KUKA KRL program: EPS_2_25694_BP03_A_20251120043254.src

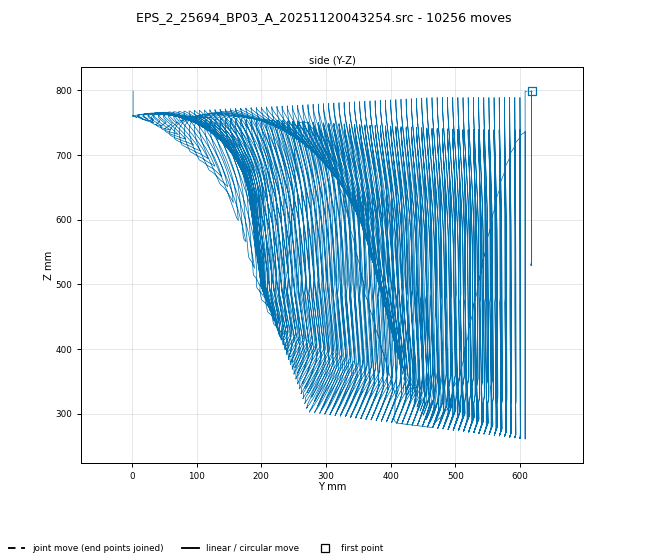
[picture p0: tool path of EPS_2_25694_BP03_A_20251120043254.src, 10256 of 10258 moves have a stored position in this frame; points joined in program order, loops and branches not executed]
&ACCESS RVP
&REL 4
&COMMENT QRS 19112012
&PARAM EDITMASK = *
DEF PART()
EXT BAS (BAS_COMMAND :IN,REAL :IN )
INT I
BAS (#INITMOV,0 )

;KUKA QRS Post kuka4.cps  Date:22-06-2017 !

File_ID=2919

QRS_PRE_INIT()

;Init var - Until changes are made in qrs_pre_init
Outlet_Square_prg=0
Inlet_1_Square_prg=0
Inlet_2_Square_prg=0
Inlet_3_Square_prg=0
Inlet_4_Square_prg=0
Inlet_5_Square_prg=0

Outlet_1={X 0.000, Y 466.000, Z 560.500, B 0.000, E1 0.000 }
Inlet_1={X 0.000, Y 466.000, Z 548.500, B 0.000, E1 90.000 }
Inlet_2={X 0.000, Y 519.840, Z 613.500, B 0.000, E1 205.000 }
Outlet_1_type=457
Inlet_1_type=381
Inlet_2_type=251
;QRS#1=Sidecore dimensions
;QRS#2=450-18" Concrete
;QRS#3=375-15" Concrete
;QRS#4=250-10" PVC SDR 35
;QRS#5=
;QRS#6=
;QRS#7=
;QRS#8=
;QRS#9=28A PSX-2
;QRS#10=24L PSX-2
;QRS#11=14M PSX
;QRS#12=
;QRS#13=
;QRS#14=
;QRS#15=
;QRS#16=1220x127x1143 3,75'
;QRS#17=EPS Height
;QRS#18=789
;QRS#19=*
;QRS#20= UPDATED VERSION 22-06-2017
;QRS#21=*
Outlet_Square=0250
Inlet_1_Square=0150
Inlet_2_Square=0100
Inlet_3_Square=0
Inlet_4_Square=0
Inlet_5_Square=0
Mill_Square=1
Outlet_Square_Prg=274
Inlet_1_Square_prg=261
Inlet_2_Square_prg=205

QRS_INIT()

$ADVANCE=5

; T1
PTP {E1 170.917,E2 170.917}
PTP {X 0,Y 617.926,A -85,B 0,C 180,E1 170.917,E2 170.917,E3 0,E4 0,E5 0,E6 0}
QRS_SPEED_INIT()
LIN {X 0,Y 617.926,Z 799,A -85,B 0,C 180,E1 170.917,E2 170.917,E3 0,E4 0,E5 0,E6 0} C_VEL
LIN {X 0,Y 617.926,Z 732.08,A -85,B 0,C 180,E1 170.917,E2 170.917} C_VEL
LIN {X 0,Y 617.926,Z 723.896,A -85,B 0,C 180,E1 170.917,E2 170.917} C_VEL
LIN {X 0,Y 617.92,Z 722.066,A -85,B 0,C 180,E1 171.177,E2 171.177} C_VEL
LIN {X 0,Y 617.969,Z 725.43,A -85,B 0,C 180,E1 171.885,E2 171.885} C_VEL
LIN {X 0,Y 617.858,Z 729.365,A -85,B 0,C 180,E1 172.817,E2 172.817} C_VEL
LIN {X 0,Y 617.844,Z 732.739,A -85,B 0,C 180,E1 173.747,E2 173.747} C_VEL
LIN {X 0,Y 617.965,Z 735.568,A -85,B 0,C 180,E1 174.678,E2 174.678} C_VEL
LIN {X 0,Y 617.921,Z 737.95,A -85,B 0,C 180,E1 175.605,E2 175.605} C_VEL
LIN {X 0,Y 617.836,Z 739.867,A -85,B 0,C 180,E1 176.531,E2 176.531} C_VEL
LIN {X 0,Y 617.889,Z 741.283,A -85,B 0,C 180,E1 177.457,E2 177.457} C_VEL
LIN {X 0,Y 617.913,Z 742.583,A -85,B 0,C 180,E1 178.844,E2 178.844} C_VEL
LIN {X 0,Y 617.836,Z 742.919,A -85,B 0,C 180,E1 179.769,E2 179.769} C_VEL
LIN {X 0,Y 617.896,Z 742.773,A -85,B 0,C 180,E1 180.693,E2 180.693} C_VEL
LIN {X 0,Y 617.953,Z 742.507,A -85,B 0,C 180,E1 181.155,E2 181.155} C_VEL
LIN {X 0,Y 617.906,Z 741.719,A -85,B 0,C 180,E1 182.08,E2 182.08} C_VEL
LIN {X 0,Y 617.845,Z 741.189,A -85,B 0,C 180,E1 182.543,E2 182.543} C_VEL
LIN {X 0,Y 617.837,Z 739.718,A -85,B 0,C 180,E1 183.469,E2 183.469} C_VEL
LIN {X 0,Y 617.952,Z 737.748,A -85,B 0,C 180,E1 184.395,E2 184.395} C_VEL
LIN {X 0,Y 617.906,Z 735.343,A -85,B 0,C 180,E1 185.323,E2 185.323} C_VEL
LIN {X 0,Y 617.823,Z 732.457,A -85,B 0,C 180,E1 186.253,E2 186.253} C_VEL
LIN {X 0,Y 617.893,Z 729.022,A -85,B 0,C 180,E1 187.183,E2 187.183} C_VEL
LIN {X 0,Y 617.971,Z 725.042,A -85,B 0,C 180,E1 188.115,E2 188.115} C_VEL
LIN {X 0,Y 617.879,Z 720.318,A -85,B 0,C 180,E1 189.086,E2 189.086} C_VEL
LIN {X 0,Y 617.904,Z 714.839,A -85,B 0,C 180,E1 190.065,E2 190.065} C_VEL
LIN {X 0,Y 617.99,Z 710.607,A -85,B 0,C 180,E1 190.75,E2 190.75} C_VEL
LIN {X 0,Y 617.939,Z 704.579,A -85,B 0,C 180,E1 191.634,E2 191.634} C_VEL
LIN {X 0,Y 617.924,Z 699.032,A -85,B 0,C 180,E1 192.373,E2 192.373} C_VEL
LIN {X 0,Y 617.977,Z 692.923,A -85,B 0,C 180,E1 193.112,E2 193.112} C_VEL
LIN {X 0,Y 617.99,Z 686.213,A -85,B 0,C 180,E1 193.854,E2 193.854} C_VEL
LIN {X 0,Y 617.953,Z 678.824,A -85,B 0,C 180,E1 194.6,E2 194.6} C_VEL
LIN {X 0,Y 617.973,Z 671.228,A -85,B 0,C 180,E1 195.296,E2 195.296} C_VEL
LIN {X 0,Y 617.987,Z 664.189,A -85,B 0,C 180,E1 195.886,E2 195.886} C_VEL
LIN {X 0,Y 617.986,Z 657.726,A -85,B 0,C 180,E1 196.388,E2 196.388} C_VEL
LIN {X 0,Y 617.976,Z 650.68,A -85,B 0,C 180,E1 196.894,E2 196.894} C_VEL
LIN {X 0,Y 617.993,Z 642.968,A -85,B 0,C 180,E1 197.402,E2 197.402} C_VEL
LIN {X 0,Y 617.989,Z 634.017,A -85,B 0,C 180,E1 197.935,E2 197.935} C_VEL
LIN {X 0,Y 618.005,Z 624.088,A -85,B 0,C 180,E1 198.462,E2 198.462} C_VEL
LIN {X 0,Y 617.991,Z 616.381,A -85,B 0,C 180,E1 198.833,E2 198.833} C_VEL
LIN {X 0,Y 617.89,Z 606.2,A -85,B 0,C 180,E1 199.269,E2 199.269} C_VEL
LIN {X 0,Y 617.965,Z 596.887,A -85,B 0,C 180,E1 199.613,E2 199.613} C_VEL
LIN {X 0,Y 617.956,Z 586.341,A -85,B 0,C 180,E1 199.95,E2 199.95} C_VEL
LIN {X 0,Y 617.862,Z 577.249,A -85,B 0,C 180,E1 200.201,E2 200.201} C_VEL
LIN {X 0,Y 617.986,Z 567.625,A -85,B 0,C 180,E1 200.414,E2 200.414} C_VEL
LIN {X 0,Y 618.002,Z 557.725,A -85,B 0,C 180,E1 200.59,E2 200.59} C_VEL
LIN {X 0,Y 617.92,Z 547.688,A -85,B 0,C 180,E1 200.731,E2 200.731} C_VEL
LIN {X 0,Y 618.031,Z 529.66,A -85,B 0,C 180,E1 201.975,E2 201.975} C_VEL
LIN {X 0,Y 618.043,Z 529.66,A -85,B 0,C 180,E1 202.525,E2 202.525} C_VEL
LIN {X 0,Y 617.459,Z 529.66,A -85,B 0,C 180,E1 205.076,E2 205.076} C_VEL
LIN {X 0,Y 617.91,Z 529.66,A -85,B 0,C 180,E1 207.635,E2 207.635} C_VEL
LIN {X 0,Y 617.392,Z 529.66,A -85,B 0,C 180,E1 210.305,E2 210.305} C_VEL
LIN {X 0,Y 617.847,Z 529.66,A -85,B 0,C 180,E1 212.995,E2 212.995} C_VEL
LIN {X 0,Y 617.717,Z 529.66,A -85,B 0,C 180,E1 214.197,E2 214.197} C_VEL
LIN {X 0,Y 617.793,Z 529.66,A -85,B 0,C 180,E1 218.704,E2 218.704} C_VEL
LIN {X 0,Y 617.441,Z 529.66,A -85,B 0,C 180,E1 221.76,E2 221.76} C_VEL
LIN {X 0,Y 617.845,Z 529.66,A -85,B 0,C 180,E1 224.904,E2 224.904} C_VEL
LIN {X 0,Y 617.793,Z 529.66,A -85,B 0,C 180,E1 228.273,E2 228.273} C_VEL
LIN {X 0,Y 617.576,Z 529.66,A -85,B 0,C 180,E1 231.28,E2 231.28} C_VEL
LIN {X 0,Y 617.602,Z 529.66,A -85,B 0,C 180,E1 231.897,E2 231.897} C_VEL
LIN {X 0,Y 617.843,Z 529.66,A -85,B 0,C 180,E1 234.203,E2 234.203} C_VEL
LIN {X 0,Y 617.363,Z 529.66,A -85,B 0,C 180,E1 236.975,E2 236.975} C_VEL
LIN {X 0,Y 617.906,Z 529.66,A -85,B 0,C 180,E1 239.723,E2 239.723} C_VEL
LIN {X 0,Y 618.083,Z 529.66,A -85,B 0,C 180,E1 244.632,E2 244.632} C_VEL
LIN {X 0,Y 617.159,Z 529.66,A -85,B 0,C 180,E1 244.911,E2 244.911} C_VEL
LIN {X 0,Y 616.927,Z 529.66,A -85,B 0,C 180,E1 244.938,E2 244.938} C_VEL
LIN {X 0,Y 617.36,Z 531.378,A -85,B 0,C 180,E1 244.996,E2 244.996} C_VEL
LIN {X 0,Y 617.708,Z 533.348,A -85,B 0,C 180,E1 245.036,E2 245.036} C_VEL
LIN {X 0,Y 617.911,Z 571.481,A -85,B 0,C 180,E1 245.532,E2 245.532} C_VEL
LIN {X 0,Y 617.861,Z 581.835,A -85,B 0,C 180,E1 245.699,E2 245.699} C_VEL
LIN {X 0,Y 617.79,Z 590.391,A -85,B 0,C 180,E1 245.865,E2 245.865} C_VEL
LIN {X 0,Y 617.893,Z 603.702,A -85,B 0,C 180,E1 246.204,E2 246.204} C_VEL
LIN {X 0,Y 617.821,Z 614.916,A -85,B 0,C 180,E1 246.539,E2 246.539} C_VEL
LIN {X 0,Y 617.932,Z 626.994,A -85,B 0,C 180,E1 246.972,E2 246.972} C_VEL
LIN {X 0,Y 617.944,Z 637.348,A -85,B 0,C 180,E1 247.392,E2 247.392} C_VEL
LIN {X 0,Y 617.878,Z 647.649,A -85,B 0,C 180,E1 247.858,E2 247.858} C_VEL
LIN {X 0,Y 617.947,Z 658.321,A -85,B 0,C 180,E1 248.405,E2 248.405} C_VEL
LIN {X 0,Y 617.967,Z 669.198,A -85,B 0,C 180,E1 249.026,E2 249.026} C_VEL
LIN {X 0,Y 617.938,Z 679.008,A -85,B 0,C 180,E1 249.643,E2 249.643} C_VEL
LIN {X 0,Y 617.951,Z 688.519,A -85,B 0,C 180,E1 250.301,E2 250.301} C_VEL
LIN {X 0,Y 617.957,Z 697.722,A -85,B 0,C 180,E1 250.999,E2 250.999} C_VEL
LIN {X 0,Y 617.967,Z 706.076,A -85,B 0,C 180,E1 251.689,E2 251.689} C_VEL
LIN {X 0,Y 617.94,Z 715.022,A -85,B 0,C 180,E1 252.496,E2 252.496} C_VEL
LIN {X 0,Y 617.892,Z 722.427,A -85,B 0,C 180,E1 253.221,E2 253.221} C_VEL
LIN {X 0,Y 617.945,Z 730.141,A -85,B 0,C 180,E1 254.048,E2 254.048} C_VEL
LIN {X 0,Y 617.967,Z 736.655,A -85,B 0,C 180,E1 254.802,E2 254.802} C_VEL
LIN {X 0,Y 617.884,Z 743.768,A -85,B 0,C 180,E1 255.696,E2 255.696} C_VEL
LIN {X 0,Y 617.874,Z 750.232,A -85,B 0,C 180,E1 256.588,E2 256.588} C_VEL
LIN {X 0,Y 617.98,Z 756.092,A -85,B 0,C 180,E1 257.48,E2 257.48} C_VEL
LIN {X 0,Y 617.887,Z 761.455,A -85,B 0,C 180,E1 258.364,E2 258.364} C_VEL
LIN {X 0,Y 617.832,Z 767.76,A -85,B 0,C 180,E1 259.541,E2 259.541} C_VEL
LIN {X 0,Y 617.909,Z 771.343,A -85,B 0,C 180,E1 260.283,E2 260.283} C_VEL
LIN {X 0,Y 617.921,Z 776.378,A -85,B 0,C 180,E1 261.453,E2 261.453} C_VEL
LIN {X 0,Y 617.825,Z 779.754,A -85,B 0,C 180,E1 262.349,E2 262.349} C_VEL
LIN {X 0,Y 617.934,Z 784.147,A -85,B 0,C 180,E1 263.747,E2 263.747} C_VEL
LIN {X 0,Y 617.912,Z 786.615,A -85,B 0,C 180,E1 264.676,E2 264.676} C_VEL
LIN {X 0,Y 617.789,Z 788.667,A -85,B 0,C 180,E1 265.603,E2 265.603} C_VEL
LIN {X 0,Y 617.809,Z 790.257,A -85,B 0,C 180,E1 266.53,E2 266.53} C_VEL
LIN {X 0,Y 617.945,Z 791.44,A -85,B 0,C 180,E1 267.456,E2 267.456} C_VEL
LIN {X 0,Y 617.797,Z 792.66,A -85,B 0,C 180,E1 268.843,E2 268.843} C_VEL
LIN {X 0,Y 617.788,Z 792.921,A -85,B 0,C 180,E1 269.768,E2 269.768} C_VEL
LIN {X 0,Y 617.983,Z 792.611,A -85,B 0,C 180,E1 271.154,E2 271.154} C_VEL
LIN {X 0,Y 617.853,Z 791.992,A -85,B 0,C 180,E1 272.08,E2 272.08} C_VEL
LIN {X 0,Y 617.854,Z 790.248,A -85,B 0,C 180,E1 273.468,E2 273.468} C_VEL
LIN {X 0,Y 617.999,Z 788.615,A -85,B 0,C 180,E1 274.393,E2 274.393} C_VEL
LIN {X 0,Y 617.855,Z 786.634,A -85,B 0,C 180,E1 275.322,E2 275.322} C_VEL
LIN {X 0,Y 617.792,Z 784.189,A -85,B 0,C 180,E1 276.252,E2 276.252} C_VEL
LIN {X 0,Y 617.955,Z 779.729,A -85,B 0,C 180,E1 277.647,E2 277.647} C_VEL
LIN {X 0,Y 617.882,Z 775.324,A -85,B 0,C 180,E1 278.801,E2 278.801} C_VEL
LIN {X 0,Y 617.827,Z 771.607,A -85,B 0,C 180,E1 279.667,E2 279.667} C_VEL
LIN {X 0,Y 617.937,Z 766.262,A -85,B 0,C 180,E1 280.75,E2 280.75} C_VEL
LIN {X 0,Y 617.943,Z 761.454,A -85,B 0,C 180,E1 281.633,E2 281.633} C_VEL
LIN {X 0,Y 617.869,Z 754.203,A -85,B 0,C 180,E1 282.817,E2 282.817} C_VEL
LIN {X 0,Y 617.947,Z 748.142,A -85,B 0,C 180,E1 283.705,E2 283.705} C_VEL
LIN {X 0,Y 617.964,Z 741.476,A -85,B 0,C 180,E1 284.599,E2 284.599} C_VEL
LIN {X 0,Y 617.886,Z 733.506,A -85,B 0,C 180,E1 285.571,E2 285.571} C_VEL
LIN {X 0,Y 617.919,Z 726.446,A -85,B 0,C 180,E1 286.357,E2 286.357} C_VEL
LIN {X 0,Y 617.968,Z 718.296,A -85,B 0,C 180,E1 287.187,E2 287.187} C_VEL
LIN {X 0,Y 617.931,Z 711.158,A -85,B 0,C 180,E1 287.863,E2 287.863} C_VEL
LIN {X 0,Y 617.922,Z 702.259,A -85,B 0,C 180,E1 288.634,E2 288.634} C_VEL
LIN {X 0,Y 617.943,Z 693.364,A -85,B 0,C 180,E1 289.339,E2 289.339} C_VEL
LIN {X 0,Y 617.96,Z 684.874,A -85,B 0,C 180,E1 289.958,E2 289.958} C_VEL
LIN {X 0,Y 617.948,Z 675.484,A -85,B 0,C 180,E1 290.586,E2 290.586} C_VEL
LIN {X 0,Y 617.918,Z 665.294,A -85,B 0,C 180,E1 291.206,E2 291.206} C_VEL
LIN {X 0,Y 617.944,Z 655.431,A -85,B 0,C 180,E1 291.748,E2 291.748} C_VEL
LIN {X 0,Y 617.958,Z 644.378,A -85,B 0,C 180,E1 292.293,E2 292.293} C_VEL
LIN {X 0,Y 617.922,Z 633.61,A -85,B 0,C 180,E1 292.767,E2 292.767} C_VEL
LIN {X 0,Y 617.804,Z 623.469,A -85,B 0,C 180,E1 293.168,E2 293.168} C_VEL
LIN {X 0,Y 617.933,Z 610.311,A -85,B 0,C 180,E1 293.6,E2 293.6} C_VEL
LIN {X 0,Y 617.911,Z 598.948,A -85,B 0,C 180,E1 293.921,E2 293.921} C_VEL
LIN {X 0,Y 617.756,Z 588.083,A -85,B 0,C 180,E1 294.183,E2 294.183} C_VEL
LIN {X 0,Y 617.908,Z 576.195,A -85,B 0,C 180,E1 294.398,E2 294.398} C_VEL
LIN {X 0,Y 617.869,Z 558.096,A -85,B 0,C 180,E1 294.647,E2 294.647} C_VEL
LIN {X 0,Y 617.639,Z 532.594,A -85,B 0,C 180,E1 294.977,E2 294.977} C_VEL
LIN {X 0,Y 616.927,Z 529.66,A -85,B 0,C 180,E1 295.061,E2 295.061} C_VEL
LIN {X 0,Y 617.143,Z 529.66,A -85,B 0,C 180,E1 295.088,E2 295.088} C_VEL
LIN {X 0,Y 618.084,Z 529.66,A -85,B 0,C 180,E1 295.366,E2 295.366} C_VEL
LIN {X 0,Y 617.906,Z 529.66,A -85,B 0,C 180,E1 300.275,E2 300.275} C_VEL
LIN {X 0,Y 617.362,Z 529.66,A -85,B 0,C 180,E1 303.022,E2 303.022} C_VEL
LIN {X 0,Y 617.841,Z 529.66,A -85,B 0,C 180,E1 305.795,E2 305.795} C_VEL
LIN {X 0,Y 617.942,Z 529.66,A -85,B 0,C 180,E1 308.691,E2 308.691} C_VEL
LIN {X 0,Y 617.455,Z 529.66,A -85,B 0,C 180,E1 311.757,E2 311.757} C_VEL
LIN {X 0,Y 617.882,Z 529.66,A -85,B 0,C 180,E1 314.898,E2 314.898} C_VEL
LIN {X 0,Y 617.778,Z 529.66,A -85,B 0,C 180,E1 318.272,E2 318.272} C_VEL
LIN {X 0,Y 617.552,Z 529.66,A -85,B 0,C 180,E1 321.278,E2 321.278} C_VEL
LIN {X 0,Y 617.581,Z 529.66,A -85,B 0,C 180,E1 321.897,E2 321.897} C_VEL
LIN {X 0,Y 617.811,Z 529.66,A -85,B 0,C 180,E1 324.202,E2 324.202} C_VEL
LIN {X 0,Y 617.353,Z 529.66,A -85,B 0,C 180,E1 326.975,E2 326.975} C_VEL
LIN {X 0,Y 617.896,Z 529.66,A -85,B 0,C 180,E1 329.723,E2 329.723} C_VEL
LIN {X 0,Y 617.434,Z 529.66,A -85,B 0,C 180,E1 332.342,E2 332.342} C_VEL
LIN {X 0,Y 617.928,Z 529.66,A -85,B 0,C 180,E1 334.945,E2 334.945} C_VEL
LIN {X 0,Y 617.462,Z 529.66,A -85,B 0,C 180,E1 337.452,E2 337.452} C_VEL
LIN {X 0,Y 617.953,Z 529.66,A -85,B 0,C 180,E1 339.952,E2 339.952} C_VEL
LIN {X 0,Y 618.034,Z 529.66,A -85,B 0,C 180,E1 343.628,E2 343.628} C_VEL
LIN {X 0,Y 618.009,Z 529.66,A -85,B 0,C 180,E1 349.544,E2 349.544} C_VEL
LIN {X 0,Y 618.004,Z 529.66,A -85,B 0,C 180,E1 354.214,E2 354.214} C_VEL
LIN {X 0,Y 618.059,Z 529.66,A -85,B 0,C 180,E1 358.845,E2 358.845} C_VEL
LIN {X 0,Y 618.056,Z 529.66,A -85,B 0,C 180,E1 363.468,E2 363.468} C_VEL
LIN {X 0,Y 618.007,Z 529.66,A -85,B 0,C 180,E1 368.114,E2 368.114} C_VEL
LIN {X 0,Y 617.998,Z 529.66,A -85,B 0,C 180,E1 372.815,E2 372.815} C_VEL
LIN {X 0,Y 617.967,Z 529.66,A -85,B 0,C 180,E1 377.606,E2 377.606} C_VEL
LIN {X 0,Y 617.769,Z 529.66,A -85,B 0,C 180,E1 378.552,E2 378.552} C_VEL
LIN {X 0,Y 617.916,Z 529.66,A -85,B 0,C 180,E1 382.53,E2 382.53} C_VEL
LIN {X 0,Y 617.427,Z 529.66,A -85,B 0,C 180,E1 385.077,E2 385.077} C_VEL
LIN {X 0,Y 617.881,Z 529.66,A -85,B 0,C 180,E1 387.637,E2 387.637} C_VEL
LIN {X 0,Y 617.377,Z 529.66,A -85,B 0,C 180,E1 390.305,E2 390.305} C_VEL
LIN {X 0,Y 617.855,Z 529.66,A -85,B 0,C 180,E1 392.994,E2 392.994} C_VEL
LIN {X 0,Y 617.713,Z 529.66,A -85,B 0,C 180,E1 394.2,E2 394.2} C_VEL
LIN {X 0,Y 617.795,Z 529.66,A -85,B 0,C 180,E1 398.704,E2 398.704} C_VEL
LIN {X 0,Y 617.422,Z 529.66,A -85,B 0,C 180,E1 401.762,E2 401.762} C_VEL
LIN {X 0,Y 617.795,Z 529.66,A -85,B 0,C 180,E1 404.908,E2 404.908} C_VEL
LIN {X 0,Y 618.001,Z 529.66,A -85,B 0,C 180,E1 409.511,E2 409.511} C_VEL
LIN {X 0,Y 617.94,Z 532.312,A -85,B 0,C 180,E1 409.607,E2 409.607} C_VEL
LIN {X 0,Y 618.041,Z 612.613,A -85,B 0,C 180,E1 410.568,E2 410.568} C_VEL
LIN {X 0,Y 617.973,Z 623.423,A -85,B 0,C 180,E1 410.768,E2 410.768} C_VEL
LIN {X 0,Y 617.981,Z 631.663,A -85,B 0,C 180,E1 410.974,E2 410.974} C_VEL
LIN {X 0,Y 617.976,Z 641.062,A -85,B 0,C 180,E1 411.264,E2 411.264} C_VEL
LIN {X 0,Y 618.033,Z 650.601,A -85,B 0,C 180,E1 411.631,E2 411.631} C_VEL
LIN {X 0,Y 618.03,Z 658.048,A -85,B 0,C 180,E1 411.966,E2 411.966} C_VEL
LIN {X 0,Y 618.018,Z 666.559,A -85,B 0,C 180,E1 412.404,E2 412.404} C_VEL
LIN {X 0,Y 618.005,Z 675.252,A -85,B 0,C 180,E1 412.927,E2 412.927} C_VEL
LIN {X 0,Y 618.018,Z 683.518,A -85,B 0,C 180,E1 413.498,E2 413.498} C_VEL
LIN {X 0,Y 617.975,Z 691.288,A -85,B 0,C 180,E1 414.112,E2 414.112} C_VEL
LIN {X 0,Y 617.978,Z 697.764,A -85,B 0,C 180,E1 414.692,E2 414.692} C_VEL
LIN {X 0,Y 617.974,Z 704.384,A -85,B 0,C 180,E1 415.356,E2 415.356} C_VEL
LIN {X 0,Y 617.999,Z 710.463,A -85,B 0,C 180,E1 416.056,E2 416.056} C_VEL
LIN {X 0,Y 617.982,Z 715.444,A -85,B 0,C 180,E1 416.696,E2 416.696} C_VEL
LIN {X 0,Y 617.936,Z 720.306,A -85,B 0,C 180,E1 417.394,E2 417.394} C_VEL
LIN {X 0,Y 617.97,Z 724.771,A -85,B 0,C 180,E1 418.136,E2 418.136} C_VEL
LIN {X 0,Y 617.977,Z 729.544,A -85,B 0,C 180,E1 419.057,E2 419.057} C_VEL
LIN {X 0,Y 617.923,Z 732.523,A -85,B 0,C 180,E1 419.726,E2 419.726} C_VEL
LIN {X 0,Y 617.935,Z 735.597,A -85,B 0,C 180,E1 420.545,E2 420.545} C_VEL
LIN {X 0,Y 618.004,Z 738.354,A -85,B 0,C 180,E1 421.473,E2 421.473} C_VEL
LIN {X 0,Y 617.93,Z 740.45,A -85,B 0,C 180,E1 422.367,E2 422.367} C_VEL
LIN {X 0,Y 617.93,Z 741.544,A -85,B 0,C 180,E1 423.017,E2 423.017} C_VEL
LIN {X 0,Y 617.982,Z 742.304,A -85,B 0,C 180,E1 423.666,E2 423.666} C_VEL
LIN {X 0,Y 617.966,Z 742.768,A -85,B 0,C 180,E1 424.308,E2 424.308} C_VEL
LIN {X 0,Y 617.895,Z 742.898,A -85,B 0,C 180,E1 425.167,E2 425.167} C_VEL
LIN {X 0,Y 617.901,Z 742.764,A -85,B 0,C 180,E1 425.638,E2 425.638} C_VEL
LIN {X 0,Y 617.982,Z 742.094,A -85,B 0,C 180,E1 426.424,E2 426.424} C_VEL
LIN {X 0,Y 617.943,Z 740.577,A -85,B 0,C 180,E1 427.472,E2 427.472} C_VEL
LIN {X 0,Y 617.91,Z 739.26,A -85,B 0,C 180,E1 428.095,E2 428.095} C_VEL
LIN {X 0,Y 617.948,Z 737.617,A -85,B 0,C 180,E1 428.718,E2 428.718} C_VEL
LIN {X 0,Y 617.983,Z 734.576,A -85,B 0,C 180,E1 429.646,E2 429.646} C_VEL
LIN {X 0,Y 617.929,Z 730.51,A -85,B 0,C 180,E1 430.652,E2 430.652} C_VEL
LIN {X 0,Y 617.977,Z 726.839,A -85,B 0,C 180,E1 431.396,E2 431.396} C_VEL
LIN {X 0,Y 617.989,Z 722.638,A -85,B 0,C 180,E1 432.135,E2 432.135} C_VEL
LIN {X 0,Y 617.964,Z 718.088,A -85,B 0,C 180,E1 432.843,E2 432.843} C_VEL
LIN {X 0,Y 617.988,Z 712.092,A -85,B 0,C 180,E1 433.655,E2 433.655} C_VEL
LIN {X 0,Y 618.005,Z 705.641,A -85,B 0,C 180,E1 434.412,E2 434.412} C_VEL
LIN {X 0,Y 617.988,Z 698.978,A -85,B 0,C 180,E1 435.103,E2 435.103} C_VEL
LIN {X 0,Y 618.01,Z 692.402,A -85,B 0,C 180,E1 435.701,E2 435.701} C_VEL
LIN {X 0,Y 618.03,Z 685.073,A -85,B 0,C 180,E1 436.297,E2 436.297} C_VEL
LIN {X 0,Y 618.02,Z 676.665,A -85,B 0,C 180,E1 436.89,E2 436.89} C_VEL
LIN {X 0,Y 618.022,Z 669.526,A -85,B 0,C 180,E1 437.335,E2 437.335} C_VEL
LIN {X 0,Y 618.037,Z 661.46,A -85,B 0,C 180,E1 437.779,E2 437.779} C_VEL
LIN {X 0,Y 618.044,Z 653.666,A -85,B 0,C 180,E1 438.148,E2 438.148} C_VEL
LIN {X 0,Y 618.031,Z 646.548,A -85,B 0,C 180,E1 438.443,E2 438.443} C_VEL
LIN {X 0,Y 617.957,Z 638.331,A -85,B 0,C 180,E1 438.736,E2 438.736} C_VEL
LIN {X 0,Y 618.024,Z 628.836,A -85,B 0,C 180,E1 439.013,E2 439.013} C_VEL
LIN {X 0,Y 617.998,Z 618.998,A -85,B 0,C 180,E1 439.233,E2 439.233} C_VEL
LIN {X 0,Y 617.95,Z 611.443,A -85,B 0,C 180,E1 439.361,E2 439.361} C_VEL
LIN {X 0,Y 617.885,Z 539.242,A -85,B 0,C 180,E1 440.223,E2 440.223} C_VEL
LIN {X 0,Y 617.181,Z 529.725,A -85,B 0,C 180,E1 440.354,E2 440.354} C_VEL
LIN {X 0,Y 617.577,Z 529.66,A -85,B 0,C 180,E1 440.412,E2 440.412} C_VEL
LIN {X 0,Y 617.76,Z 529.66,A -85,B 0,C 180,E1 441.273,E2 441.273} C_VEL
LIN {X 0,Y 618.047,Z 529.66,A -85,B 0,C 180,E1 446.533,E2 446.533} C_VEL
LIN {X 0,Y 618.065,Z 529.66,A -85,B 0,C 180,E1 451.156,E2 451.156} C_VEL
LIN {X 0,Y 618.057,Z 529.66,A -85,B 0,C 180,E1 455.787,E2 455.787} C_VEL
LIN {X 0,Y 617.974,Z 529.66,A -85,B 0,C 180,E1 460.457,E2 460.457} C_VEL
LIN {X 0,Y 617.948,Z 529.66,A -85,B 0,C 180,E1 465.199,E2 465.199} C_VEL
LIN {X 0,Y 617.954,Z 529.66,A -85,B 0,C 180,E1 470.049,E2 470.049} C_VEL
LIN {X 0,Y 617.465,Z 529.66,A -85,B 0,C 180,E1 472.548,E2 472.548} C_VEL
LIN {X 0,Y 617.908,Z 529.66,A -85,B 0,C 180,E1 475.057,E2 475.057} C_VEL
LIN {X 0,Y 617.411,Z 529.66,A -85,B 0,C 180,E1 477.66,E2 477.66} C_VEL
LIN {X 0,Y 617.872,Z 529.66,A -85,B 0,C 180,E1 480.279,E2 480.279} C_VEL
LIN {X 0,Y 617.352,Z 529.66,A -85,B 0,C 180,E1 483.025,E2 483.025} C_VEL
LIN {X 0,Y 617.837,Z 529.66,A -85,B 0,C 180,E1 485.797,E2 485.797} C_VEL
LIN {X 0,Y 617.931,Z 529.66,A -85,B 0,C 180,E1 488.694,E2 488.694} C_VEL
LIN {X 0,Y 617.447,Z 529.66,A -85,B 0,C 180,E1 491.76,E2 491.76} C_VEL
LIN {X 0,Y 617.885,Z 529.66,A -85,B 0,C 180,E1 494.901,E2 494.901} C_VEL
LIN {X 0,Y 617.791,Z 529.66,A -85,B 0,C 180,E1 498.273,E2 498.273} C_VEL
LIN {X 0,Y 617.548,Z 529.66,A -85,B 0,C 180,E1 501.278,E2 501.278} C_VEL
LIN {X 0,Y 617.791,Z 529.66,A -85,B 0,C 180,E1 504.2,E2 504.2} C_VEL
LIN {X 0,Y 617.319,Z 529.66,A -85,B 0,C 180,E1 506.973,E2 506.973} C_VEL
LIN {X 0,Y 617.869,Z 529.66,A -85,B 0,C 180,E1 509.721,E2 509.721} C_VEL
LIN {X 0,Y 617.427,Z 529.66,A -85,B 0,C 180,E1 512.341,E2 512.341} C_VEL
LIN {X 0,Y 617.967,Z 529.66,A -85,B 0,C 180,E1 514.946,E2 514.946} C_VEL
LIN {X 0,Y 617.999,Z 529.66,A -85,B 0,C 180,E1 518.516,E2 518.516} C_VEL
LIN {X 0,Y 617.886,Z 529.66,A -85,B 0,C 180,E1 518.873,E2 518.873} C_VEL
LIN {X 0,Y 617.56,Z 529.66,A -85,B 0,C 180,E1 518.94,E2 518.94} C_VEL
LIN {X 0,Y 617.895,Z 556.607,A -85,B 0,C 180,E1 519.3,E2 519.3} C_VEL
LIN {X 0,Y 617.852,Z 566.901,A -85,B 0,C 180,E1 519.478,E2 519.478} C_VEL
LIN {X 0,Y 617.971,Z 576.957,A -85,B 0,C 180,E1 519.706,E2 519.706} C_VEL
LIN {X 0,Y 618.004,Z 588.92,A -85,B 0,C 180,E1 520.035,E2 520.035} C_VEL
LIN {X 0,Y 617.887,Z 600.655,A -85,B 0,C 180,E1 520.427,E2 520.427} C_VEL
LIN {X 0,Y 617.99,Z 610.527,A -85,B 0,C 180,E1 520.821,E2 520.821} C_VEL
LIN {X 0,Y 617.998,Z 620.131,A -85,B 0,C 180,E1 521.253,E2 521.253} C_VEL
LIN {X 0,Y 617.971,Z 629.635,A -85,B 0,C 180,E1 521.734,E2 521.734} C_VEL
LIN {X 0,Y 617.967,Z 637.838,A -85,B 0,C 180,E1 522.196,E2 522.196} C_VEL
LIN {X 0,Y 617.976,Z 646.385,A -85,B 0,C 180,E1 522.728,E2 522.728} C_VEL
LIN {X 0,Y 617.991,Z 654.494,A -85,B 0,C 180,E1 523.285,E2 523.285} C_VEL
LIN {X 0,Y 617.973,Z 662.196,A -85,B 0,C 180,E1 523.864,E2 523.864} C_VEL
LIN {X 0,Y 617.946,Z 669.992,A -85,B 0,C 180,E1 524.505,E2 524.505} C_VEL
LIN {X 0,Y 617.932,Z 676.637,A -85,B 0,C 180,E1 525.101,E2 525.101} C_VEL
LIN {X 0,Y 617.982,Z 682.778,A -85,B 0,C 180,E1 525.699,E2 525.699} C_VEL
LIN {X 0,Y 617.965,Z 689.783,A -85,B 0,C 180,E1 526.443,E2 526.443} C_VEL
LIN {X 0,Y 617.92,Z 696.166,A -85,B 0,C 180,E1 527.183,E2 527.183} C_VEL
LIN {X 0,Y 617.927,Z 701.976,A -85,B 0,C 180,E1 527.923,E2 527.923} C_VEL
LIN {X 0,Y 617.977,Z 707.265,A -85,B 0,C 180,E1 528.661,E2 528.661} C_VEL
LIN {X 0,Y 617.946,Z 711.21,A -85,B 0,C 180,E1 529.249,E2 529.249} C_VEL
LIN {X 0,Y 617.864,Z 717.562,A -85,B 0,C 180,E1 530.318,E2 530.318} C_VEL
LIN {X 0,Y 617.907,Z 721.666,A -85,B 0,C 180,E1 531.094,E2 531.094} C_VEL
LIN {X 0,Y 617.92,Z 722.066,A -85,B 0,C 180,E1 531.177,E2 531.177} C_VEL
LIN {X 0,Y 617.94,Z 723.893,A -85,B 0,C 180,E1 531.287,E2 531.287} C_VEL
LIN {X 0,Y 617.94,Z 799,A -85,B 0,C 180,E1 531.287,E2 531.287} C_VEL
LIN {X 0,Y 617.94,Z 799,A -85,B 0,C 180,E1 531.287,E2 531.287}

QRS_NEXT_CUT()
PTP {E1 536.874,E2 536.874}
PTP {X 0,Y 607.926,A -85,B 0,C 180,E1 536.874,E2 536.874,E3 0,E4 0,E5 0,E6 0}
QRS_SPEED_INIT()
LIN {X 0,Y 607.926,Z 799,A -85,B 0,C 180,E1 536.874,E2 536.874,E3 0,E4 0,E5 0,E6 0} C_VEL
LIN {X 0,Y 607.926,Z 746.583,A -85,B 0,C 180,E1 536.874,E2 536.874} C_VEL
LIN {X 0,Y 607.926,Z 738.171,A -85,B 0,C 180,E1 536.874,E2 536.874} C_VEL
LIN {X 0,Y 607.916,Z 736.195,A -85,B 0,C 180,E1 536.715,E2 536.715} C_VEL
LIN {X 0,Y 607.917,Z 732.197,A -85,B 0,C 180,E1 534.904,E2 534.904} C_VEL
LIN {X 0,Y 607.91,Z 726.378,A -85,B 0,C 180,E1 533.104,E2 533.104} C_VEL
LIN {X 0,Y 607.913,Z 719.011,A -85,B 0,C 180,E1 531.392,E2 531.392} C_VEL
LIN {X 0,Y 607.912,Z 710.203,A -85,B 0,C 180,E1 529.768,E2 529.768} C_VEL
LIN {X 0,Y 607.913,Z 699.301,A -85,B 0,C 180,E1 528.132,E2 528.132} C_VEL
LIN {X 0,Y 607.913,Z 686.828,A -85,B 0,C 180,E1 526.59,E2 526.59} C_VEL
LIN {X 0,Y 607.915,Z 673.153,A -85,B 0,C 180,E1 525.181,E2 525.181} C_VEL
LIN {X 0,Y 607.917,Z 658.405,A -85,B 0,C 180,E1 523.91,E2 523.91} C_VEL
LIN {X 0,Y 607.919,Z 642.683,A -85,B 0,C 180,E1 522.779,E2 522.779} C_VEL
LIN {X 0,Y 607.913,Z 626.024,A -85,B 0,C 180,E1 521.79,E2 521.79} C_VEL
LIN {X 0,Y 607.915,Z 608.442,A -85,B 0,C 180,E1 520.944,E2 520.944} C_VEL
LIN {X 0,Y 607.91,Z 590.522,A -85,B 0,C 180,E1 520.27,E2 520.27} C_VEL
LIN {X 0,Y 607.91,Z 572.648,A -85,B 0,C 180,E1 519.768,E2 519.768} C_VEL
LIN {X 0,Y 607.915,Z 554.05,A -85,B 0,C 180,E1 519.417,E2 519.417} C_VEL
LIN {X 0,Y 607.913,Z 342.093,A -85,B 0,C 180,E1 516.75,E2 516.75} C_VEL
LIN {X 0,Y 607.872,Z 299.576,A -85,B 0,C 180,E1 513.695,E2 513.695} C_VEL
LIN {X 0,Y 607.918,Z 261.354,A -85,B 0,C 180,E1 510.867,E2 510.867} C_VEL
LIN {X 0,Y 607.912,Z 260.757,A -85,B 0,C 180,E1 510.65,E2 510.65} C_VEL
LIN {X 0,Y 607.867,Z 260.764,A -85,B 0,C 180,E1 507.546,E2 507.546} C_VEL
LIN {X 0,Y 607.884,Z 260.759,A -85,B 0,C 180,E1 504.273,E2 504.273} C_VEL
LIN {X 0,Y 607.911,Z 260.765,A -85,B 0,C 180,E1 501.196,E2 501.196} C_VEL
LIN {X 0,Y 607.881,Z 260.759,A -85,B 0,C 180,E1 497.975,E2 497.975} C_VEL
LIN {X 0,Y 607.906,Z 260.759,A -85,B 0,C 180,E1 494.855,E2 494.855} C_VEL
LIN {X 0,Y 607.896,Z 260.762,A -85,B 0,C 180,E1 491.691,E2 491.691} C_VEL
LIN {X 0,Y 607.919,Z 260.754,A -85,B 0,C 180,E1 488.441,E2 488.441} C_VEL
LIN {X 0,Y 607.897,Z 260.762,A -85,B 0,C 180,E1 485.168,E2 485.168} C_VEL
LIN {X 0,Y 607.907,Z 260.758,A -85,B 0,C 180,E1 482.091,E2 482.091} C_VEL
LIN {X 0,Y 607.882,Z 260.759,A -85,B 0,C 180,E1 478.92,E2 478.92} C_VEL
LIN {X 0,Y 607.913,Z 260.765,A -85,B 0,C 180,E1 475.736,E2 475.736} C_VEL
LIN {X 0,Y 607.88,Z 260.759,A -85,B 0,C 180,E1 472.638,E2 472.638} C_VEL
LIN {X 0,Y 607.875,Z 260.763,A -85,B 0,C 180,E1 469.407,E2 469.407} C_VEL
LIN {X 0,Y 607.886,Z 260.76,A -85,B 0,C 180,E1 466.435,E2 466.435} C_VEL
LIN {X 0,Y 607.853,Z 260.764,A -85,B 0,C 180,E1 463.315,E2 463.315} C_VEL
LIN {X 0,Y 607.88,Z 260.763,A -85,B 0,C 180,E1 460.385,E2 460.385} C_VEL
LIN {X 0,Y 607.835,Z 260.767,A -85,B 0,C 180,E1 457.278,E2 457.278} C_VEL
LIN {X 0,Y 607.89,Z 260.966,A -85,B 0,C 180,E1 456.257,E2 456.257} C_VEL
LIN {X 0,Y 607.917,Z 266.861,A -85,B 0,C 180,E1 455.759,E2 455.759} C_VEL
LIN {X 0,Y 607.901,Z 307.026,A -85,B 0,C 180,E1 452.688,E2 452.688} C_VEL
LIN {X 0,Y 607.906,Z 348.222,A -85,B 0,C 180,E1 449.624,E2 449.624} C_VEL
LIN {X 0,Y 607.895,Z 390.467,A -85,B 0,C 180,E1 446.559,E2 446.559} C_VEL
LIN {X 0,Y 607.879,Z 435.108,A -85,B 0,C 180,E1 443.39,E2 443.39} C_VEL
LIN {X 0,Y 607.906,Z 472.483,A -85,B 0,C 180,E1 440.797,E2 440.797} C_VEL
LIN {X 0,Y 607.898,Z 614.271,A -85,B 0,C 180,E1 439.072,E2 439.072} C_VEL
LIN {X 0,Y 607.919,Z 631.005,A -85,B 0,C 180,E1 438.69,E2 438.69} C_VEL
LIN {X 0,Y 607.916,Z 645.866,A -85,B 0,C 180,E1 438.185,E2 438.185} C_VEL
LIN {X 0,Y 607.916,Z 660.472,A -85,B 0,C 180,E1 437.51,E2 437.51} C_VEL
LIN {X 0,Y 607.918,Z 675.006,A -85,B 0,C 180,E1 436.64,E2 436.64} C_VEL
LIN {X 0,Y 607.918,Z 687.294,A -85,B 0,C 180,E1 435.718,E2 435.718} C_VEL
LIN {X 0,Y 607.918,Z 699.759,A -85,B 0,C 180,E1 434.548,E2 434.548} C_VEL
LIN {X 0,Y 607.917,Z 709.872,A -85,B 0,C 180,E1 433.372,E2 433.372} C_VEL
LIN {X 0,Y 607.917,Z 719.257,A -85,B 0,C 180,E1 431.99,E2 431.99} C_VEL
LIN {X 0,Y 607.917,Z 726.624,A -85,B 0,C 180,E1 430.597,E2 430.597} C_VEL
LIN {X 0,Y 607.918,Z 732.436,A -85,B 0,C 180,E1 429.091,E2 429.091} C_VEL
LIN {X 0,Y 607.919,Z 736.408,A -85,B 0,C 180,E1 427.57,E2 427.57} C_VEL
LIN {X 0,Y 607.917,Z 738.54,A -85,B 0,C 180,E1 426.032,E2 426.032} C_VEL
LIN {X 0,Y 607.916,Z 738.894,A -85,B 0,C 180,E1 424.476,E2 424.476} C_VEL
LIN {X 0,Y 607.914,Z 737.56,A -85,B 0,C 180,E1 423.004,E2 423.004} C_VEL
LIN {X 0,Y 607.916,Z 734.271,A -85,B 0,C 180,E1 421.437,E2 421.437} C_VEL
LIN {X 0,Y 607.914,Z 729.539,A -85,B 0,C 180,E1 420.002,E2 420.002} C_VEL
LIN {X 0,Y 607.915,Z 722.969,A -85,B 0,C 180,E1 418.577,E2 418.577} C_VEL
LIN {X 0,Y 607.919,Z 714.179,A -85,B 0,C 180,E1 417.13,E2 417.13} C_VEL
LIN {X 0,Y 607.917,Z 704.536,A -85,B 0,C 180,E1 415.887,E2 415.887} C_VEL
LIN {X 0,Y 607.918,Z 692.695,A -85,B 0,C 180,E1 414.666,E2 414.666} C_VEL
LIN {X 0,Y 607.918,Z 680.197,A -85,B 0,C 180,E1 413.637,E2 413.637} C_VEL
LIN {X 0,Y 607.906,Z 665.842,A -85,B 0,C 180,E1 412.694,E2 412.694} C_VEL
LIN {X 0,Y 607.904,Z 651.24,A -85,B 0,C 180,E1 411.953,E2 411.953} C_VEL
LIN {X 0,Y 607.917,Z 635.281,A -85,B 0,C 180,E1 411.348,E2 411.348} C_VEL
LIN {X 0,Y 607.896,Z 619.814,A -85,B 0,C 180,E1 410.941,E2 410.941} C_VEL
LIN {X 0,Y 607.871,Z 600.343,A -85,B 0,C 180,E1 410.652,E2 410.652} C_VEL
LIN {X 0,Y 607.901,Z 472.16,A -85,B 0,C 180,E1 409.1,E2 409.1} C_VEL
LIN {X 0,Y 607.844,Z 432.037,A -85,B 0,C 180,E1 406.303,E2 406.303} C_VEL
LIN {X 0,Y 607.882,Z 388.77,A -85,B 0,C 180,E1 403.228,E2 403.228} C_VEL
LIN {X 0,Y 607.899,Z 347.838,A -85,B 0,C 180,E1 400.257,E2 400.257} C_VEL
LIN {X 0,Y 607.913,Z 306.577,A -85,B 0,C 180,E1 397.189,E2 397.189} C_VEL
LIN {X 0,Y 607.919,Z 265.74,A -85,B 0,C 180,E1 394.064,E2 394.064} C_VEL
LIN {X 0,Y 607.913,Z 260.992,A -85,B 0,C 180,E1 393.661,E2 393.661} C_VEL
LIN {X 0,Y 607.864,Z 260.761,A -85,B 0,C 180,E1 390.657,E2 390.657} C_VEL
LIN {X 0,Y 607.915,Z 260.761,A -85,B 0,C 180,E1 387.566,E2 387.566} C_VEL
LIN {X 0,Y 607.864,Z 260.761,A -85,B 0,C 180,E1 384.489,E2 384.489} C_VEL
LIN {X 0,Y 607.915,Z 260.758,A -85,B 0,C 180,E1 381.315,E2 381.315} C_VEL
LIN {X 0,Y 607.871,Z 260.762,A -85,B 0,C 180,E1 378.212,E2 378.212} C_VEL
LIN {X 0,Y 607.895,Z 260.757,A -85,B 0,C 180,E1 374.966,E2 374.966} C_VEL
LIN {X 0,Y 607.892,Z 260.764,A -85,B 0,C 180,E1 371.865,E2 371.865} C_VEL
LIN {X 0,Y 607.874,Z 260.759,A -85,B 0,C 180,E1 368.609,E2 368.609} C_VEL
LIN {X 0,Y 607.911,Z 260.766,A -85,B 0,C 180,E1 365.569,E2 365.569} C_VEL
LIN {X 0,Y 607.871,Z 260.759,A -85,B 0,C 180,E1 362.451,E2 362.451} C_VEL
LIN {X 0,Y 607.914,Z 260.762,A -85,B 0,C 180,E1 359.341,E2 359.341} C_VEL
LIN {X 0,Y 607.87,Z 260.76,A -85,B 0,C 180,E1 356.228,E2 356.228} C_VEL
LIN {X 0,Y 607.911,Z 260.759,A -85,B 0,C 180,E1 353.104,E2 353.104} C_VEL
LIN {X 0,Y 607.872,Z 260.761,A -85,B 0,C 180,E1 350.055,E2 350.055} C_VEL
LIN {X 0,Y 607.915,Z 260.756,A -85,B 0,C 180,E1 346.818,E2 346.818} C_VEL
LIN {X 0,Y 607.89,Z 260.763,A -85,B 0,C 180,E1 343.665,E2 343.665} C_VEL
LIN {X 0,Y 607.882,Z 260.758,A -85,B 0,C 180,E1 340.395,E2 340.395} C_VEL
LIN {X 0,Y 607.916,Z 260.764,A -85,B 0,C 180,E1 337.263,E2 337.263} C_VEL
LIN {X 0,Y 607.875,Z 260.759,A -85,B 0,C 180,E1 334.119,E2 334.119} C_VEL
LIN {X 0,Y 607.911,Z 260.76,A -85,B 0,C 180,E1 330.975,E2 330.975} C_VEL
LIN {X 0,Y 607.875,Z 260.76,A -85,B 0,C 180,E1 327.894,E2 327.894} C_VEL
LIN {X 0,Y 607.914,Z 260.757,A -85,B 0,C 180,E1 324.739,E2 324.739} C_VEL
LIN {X 0,Y 607.88,Z 260.761,A -85,B 0,C 180,E1 321.677,E2 321.677} C_VEL
LIN {X 0,Y 607.905,Z 260.756,A -85,B 0,C 180,E1 318.447,E2 318.447} C_VEL
LIN {X 0,Y 607.908,Z 260.764,A -85,B 0,C 180,E1 315.255,E2 315.255} C_VEL
LIN {X 0,Y 607.882,Z 260.758,A -85,B 0,C 180,E1 312.022,E2 312.022} C_VEL
LIN {X 0,Y 607.912,Z 260.762,A -85,B 0,C 180,E1 308.922,E2 308.922} C_VEL
LIN {X 0,Y 607.878,Z 260.757,A -85,B 0,C 180,E1 305.816,E2 305.816} C_VEL
LIN {X 0,Y 607.909,Z 260.758,A -85,B 0,C 180,E1 302.758,E2 302.758} C_VEL
LIN {X 0,Y 607.901,Z 261.045,A -85,B 0,C 180,E1 301.19,E2 301.19} C_VEL
LIN {X 0,Y 607.917,Z 270.434,A -85,B 0,C 180,E1 300.544,E2 300.544} C_VEL
LIN {X 0,Y 607.883,Z 315.134,A -85,B 0,C 180,E1 297.7,E2 297.7} C_VEL
LIN {X 0,Y 607.916,Z 528.002,A -85,B 0,C 180,E1 294.938,E2 294.938} C_VEL
LIN {X 0,Y 607.917,Z 577.773,A -85,B 0,C 180,E1 294.278,E2 294.278} C_VEL
LIN {X 0,Y 607.906,Z 597.727,A -85,B 0,C 180,E1 293.84,E2 293.84} C_VEL
LIN {X 0,Y 607.911,Z 617.08,A -85,B 0,C 180,E1 293.248,E2 293.248} C_VEL
LIN {X 0,Y 607.916,Z 636.502,A -85,B 0,C 180,E1 292.482,E2 292.482} C_VEL
LIN {X 0,Y 607.919,Z 655.181,A -85,B 0,C 180,E1 291.566,E2 291.566} C_VEL
LIN {X 0,Y 607.917,Z 673.777,A -85,B 0,C 180,E1 290.456,E2 290.456} C_VEL
LIN {X 0,Y 607.915,Z 691.264,A -85,B 0,C 180,E1 289.204,E2 289.204} C_VEL
LIN {X 0,Y 607.914,Z 707.171,A -85,B 0,C 180,E1 287.862,E2 287.862} C_VEL
LIN {X 0,Y 607.917,Z 721.68,A -85,B 0,C 180,E1 286.432,E2 286.432} C_VEL
LIN {X 0,Y 607.909,Z 735.27,A -85,B 0,C 180,E1 284.866,E2 284.866} C_VEL
LIN {X 0,Y 607.906,Z 747.75,A -85,B 0,C 180,E1 283.171,E2 283.171} C_VEL
LIN {X 0,Y 607.905,Z 758.257,A -85,B 0,C 180,E1 281.478,E2 281.478} C_VEL
LIN {X 0,Y 607.912,Z 767.565,A -85,B 0,C 180,E1 279.657,E2 279.657} C_VEL
LIN {X 0,Y 607.914,Z 774.977,A -85,B 0,C 180,E1 277.845,E2 277.845} C_VEL
LIN {X 0,Y 607.918,Z 780.991,A -85,B 0,C 180,E1 275.946,E2 275.946} C_VEL
LIN {X 0,Y 607.916,Z 785.294,A -85,B 0,C 180,E1 274.054,E2 274.054} C_VEL
LIN {X 0,Y 607.914,Z 788.04,A -85,B 0,C 180,E1 272.073,E2 272.073} C_VEL
LIN {X 0,Y 607.912,Z 788.984,A -85,B 0,C 180,E1 270.093,E2 270.093} C_VEL
LIN {X 0,Y 607.91,Z 788.239,A -85,B 0,C 180,E1 268.208,E2 268.208} C_VEL
LIN {X 0,Y 607.915,Z 785.764,A -85,B 0,C 180,E1 266.227,E2 266.227} C_VEL
LIN {X 0,Y 607.914,Z 781.492,A -85,B 0,C 180,E1 264.241,E2 264.241} C_VEL
LIN {X 0,Y 607.913,Z 776.031,A -85,B 0,C 180,E1 262.438,E2 262.438} C_VEL
LIN {X 0,Y 607.911,Z 768.837,A -85,B 0,C 180,E1 260.628,E2 260.628} C_VEL
LIN {X 0,Y 607.909,Z 760.319,A -85,B 0,C 180,E1 258.904,E2 258.904} C_VEL
LIN {X 0,Y 607.914,Z 749.368,A -85,B 0,C 180,E1 257.074,E2 257.074} C_VEL
LIN {X 0,Y 607.911,Z 737.579,A -85,B 0,C 180,E1 255.424,E2 255.424} C_VEL
LIN {X 0,Y 607.918,Z 724.302,A -85,B 0,C 180,E1 253.846,E2 253.846} C_VEL
LIN {X 0,Y 607.916,Z 709.355,A -85,B 0,C 180,E1 252.334,E2 252.334} C_VEL
LIN {X 0,Y 607.914,Z 692.556,A -85,B 0,C 180,E1 250.894,E2 250.894} C_VEL
LIN {X 0,Y 607.916,Z 674.521,A -85,B 0,C 180,E1 249.592,E2 249.592} C_VEL
LIN {X 0,Y 607.919,Z 656.038,A -85,B 0,C 180,E1 248.482,E2 248.482} C_VEL
LIN {X 0,Y 607.916,Z 637.586,A -85,B 0,C 180,E1 247.568,E2 247.568} C_VEL
LIN {X 0,Y 607.909,Z 618.324,A -85,B 0,C 180,E1 246.795,E2 246.795} C_VEL
LIN {X 0,Y 607.906,Z 598.676,A -85,B 0,C 180,E1 246.184,E2 246.184} C_VEL
LIN {X 0,Y 607.918,Z 578.992,A -85,B 0,C 180,E1 245.746,E2 245.746} C_VEL
LIN {X 0,Y 607.91,Z 541.04,A -85,B 0,C 180,E1 245.228,E2 245.228} C_VEL
LIN {X 0,Y 607.883,Z 316.158,A -85,B 0,C 180,E1 242.324,E2 242.324} C_VEL
LIN {X 0,Y 607.885,Z 313.372,A -85,B 0,C 180,E1 242.196,E2 242.196} C_VEL
LIN {X 0,Y 607.918,Z 267.016,A -85,B 0,C 180,E1 239.235,E2 239.235} C_VEL
LIN {X 0,Y 607.903,Z 261.097,A -85,B 0,C 180,E1 238.822,E2 238.822} C_VEL
LIN {X 0,Y 607.884,Z 260.755,A -85,B 0,C 180,E1 238.073,E2 238.073} C_VEL
LIN {X 0,Y 607.904,Z 260.764,A -85,B 0,C 180,E1 234.83,E2 234.83} C_VEL
LIN {X 0,Y 607.919,Z 260.756,A -85,B 0,C 180,E1 231.559,E2 231.559} C_VEL
LIN {X 0,Y 607.873,Z 260.761,A -85,B 0,C 180,E1 228.354,E2 228.354} C_VEL
LIN {X 0,Y 607.913,Z 260.76,A -85,B 0,C 180,E1 225.255,E2 225.255} C_VEL
LIN {X 0,Y 607.868,Z 260.76,A -85,B 0,C 180,E1 222.152,E2 222.152} C_VEL
LIN {X 0,Y 607.917,Z 260.764,A -85,B 0,C 180,E1 219.045,E2 219.045} C_VEL
LIN {X 0,Y 607.867,Z 260.76,A -85,B 0,C 180,E1 215.959,E2 215.959} C_VEL
LIN {X 0,Y 607.894,Z 260.765,A -85,B 0,C 180,E1 212.761,E2 212.761} C_VEL
LIN {X 0,Y 607.875,Z 260.757,A -85,B 0,C 180,E1 209.717,E2 209.717} C_VEL
LIN {X 0,Y 607.917,Z 261.074,A -85,B 0,C 180,E1 209.079,E2 209.079} C_VEL
LIN {X 0,Y 607.882,Z 296.062,A -85,B 0,C 180,E1 206.471,E2 206.471} C_VEL
LIN {X 0,Y 607.915,Z 339.268,A -85,B 0,C 180,E1 203.352,E2 203.352} C_VEL
LIN {X 0,Y 607.913,Z 342.484,A -85,B 0,C 180,E1 203.147,E2 203.147} C_VEL
LIN {X 0,Y 607.914,Z 559.808,A -85,B 0,C 180,E1 200.407,E2 200.407} C_VEL
LIN {X 0,Y 607.914,Z 579.217,A -85,B 0,C 180,E1 199.98,E2 199.98} C_VEL
LIN {X 0,Y 607.914,Z 597.431,A -85,B 0,C 180,E1 199.404,E2 199.404} C_VEL
LIN {X 0,Y 607.915,Z 615.767,A -85,B 0,C 180,E1 198.639,E2 198.639} C_VEL
LIN {X 0,Y 607.918,Z 633.298,A -85,B 0,C 180,E1 197.714,E2 197.714} C_VEL
LIN {X 0,Y 607.915,Z 650.04,A -85,B 0,C 180,E1 196.629,E2 196.629} C_VEL
LIN {X 0,Y 607.917,Z 665.659,A -85,B 0,C 180,E1 195.404,E2 195.404} C_VEL
LIN {X 0,Y 607.915,Z 679.684,A -85,B 0,C 180,E1 194.088,E2 194.088} C_VEL
LIN {X 0,Y 607.915,Z 692.662,A -85,B 0,C 180,E1 192.635,E2 192.635} C_VEL
LIN {X 0,Y 607.917,Z 704.133,A -85,B 0,C 180,E1 191.095,E2 191.095} C_VEL
LIN {X 0,Y 607.911,Z 714.103,A -85,B 0,C 180,E1 189.466,E2 189.466} C_VEL
LIN {X 0,Y 607.912,Z 722.146,A -85,B 0,C 180,E1 187.846,E2 187.846} C_VEL
LIN {X 0,Y 607.91,Z 728.788,A -85,B 0,C 180,E1 186.137,E2 186.137} C_VEL
LIN {X 0,Y 607.905,Z 733.703,A -85,B 0,C 180,E1 184.433,E2 184.433} C_VEL
LIN {X 0,Y 607.908,Z 737.107,A -85,B 0,C 180,E1 182.639,E2 182.639} C_VEL
LIN {X 0,Y 607.917,Z 738.818,A -85,B 0,C 180,E1 180.754,E2 180.754} C_VEL
LIN {X 0,Y 607.915,Z 738.727,A -85,B 0,C 180,E1 178.963,E2 178.963} C_VEL
LIN {X 0,Y 607.912,Z 736.955,A -85,B 0,C 180,E1 177.171,E2 177.171} C_VEL
LIN {X 0,Y 607.916,Z 736.195,A -85,B 0,C 180,E1 176.715,E2 176.715} C_VEL
LIN {X 0,Y 606.897,Z 734.89,A -85,B 0,C 180,E1 175.999,E2 175.999} C_VEL
LIN {X 0,Y 601.771,Z 731.347,A -85,B 0,C 180,E1 174.518,E2 174.518} C_VEL
LIN {X 0,Y 600.007,Z 728.896,A -85,B 0,C 180,E1 173.716,E2 173.716} C_VEL
LIN {X 0,Y 599.918,Z 728.211,A -85,B 0,C 180,E1 173.514,E2 173.514} C_VEL
LIN {X 0,Y 599.921,Z 721.302,A -85,B 0,C 180,E1 171.759,E2 171.759} C_VEL
LIN {X 0,Y 599.942,Z 712.5,A -85,B 0,C 180,E1 170.018,E2 170.018} C_VEL
LIN {X 0,Y 599.964,Z 702.139,A -85,B 0,C 180,E1 168.366,E2 168.366} C_VEL
LIN {X 0,Y 600.005,Z 690.217,A -85,B 0,C 180,E1 166.803,E2 166.803} C_VEL
LIN {X 0,Y 600.044,Z 676.686,A -85,B 0,C 180,E1 165.328,E2 165.328} C_VEL
LIN {X 0,Y 600.096,Z 662.408,A -85,B 0,C 180,E1 164.025,E2 164.025} C_VEL
LIN {X 0,Y 600.153,Z 647.039,A -85,B 0,C 180,E1 162.849,E2 162.849} C_VEL
LIN {X 0,Y 600.218,Z 630.474,A -85,B 0,C 180,E1 161.799,E2 161.799} C_VEL
LIN {X 0,Y 600.273,Z 614.032,A -85,B 0,C 180,E1 160.945,E2 160.945} C_VEL
LIN {X 0,Y 600.329,Z 595.811,A -85,B 0,C 180,E1 160.193,E2 160.193} C_VEL
LIN {X 0,Y 600.38,Z 576.816,A -85,B 0,C 180,E1 159.606,E2 159.606} C_VEL
LIN {X 0,Y 600.415,Z 557.875,A -85,B 0,C 180,E1 159.205,E2 159.205} C_VEL
LIN {X 0,Y 600.429,Z 342.582,A -85,B 0,C 180,E1 156.459,E2 156.459} C_VEL
LIN {X 0,Y 600.422,Z 301.598,A -85,B 0,C 180,E1 153.494,E2 153.494} C_VEL
LIN {X 0,Y 600.567,Z 263.941,A -85,B 0,C 180,E1 150.68,E2 150.68} C_VEL
LIN {X 0,Y 599.967,Z 261.874,A -85,B 0,C 180,E1 150.442,E2 150.442} C_VEL
LIN {X 0,Y 599.936,Z 261.754,A -85,B 0,C 180,E1 147.43,E2 147.43} C_VEL
LIN {X 0,Y 599.94,Z 261.748,A -85,B 0,C 180,E1 144.198,E2 144.198} C_VEL
LIN {X 0,Y 599.974,Z 261.753,A -85,B 0,C 180,E1 141.077,E2 141.077} C_VEL
LIN {X 0,Y 599.942,Z 261.749,A -85,B 0,C 180,E1 137.871,E2 137.871} C_VEL
LIN {X 0,Y 599.97,Z 261.746,A -85,B 0,C 180,E1 134.691,E2 134.691} C_VEL
LIN {X 0,Y 599.975,Z 261.753,A -85,B 0,C 180,E1 131.415,E2 131.415} C_VEL
LIN {X 0,Y 599.961,Z 261.746,A -85,B 0,C 180,E1 128.13,E2 128.13} C_VEL
LIN {X 0,Y 599.953,Z 261.749,A -85,B 0,C 180,E1 124.981,E2 124.981} C_VEL
LIN {X 0,Y 599.97,Z 261.751,A -85,B 0,C 180,E1 121.778,E2 121.778} C_VEL
LIN {X 0,Y 599.958,Z 261.745,A -85,B 0,C 180,E1 118.564,E2 118.564} C_VEL
LIN {X 0,Y 599.942,Z 261.75,A -85,B 0,C 180,E1 115.256,E2 115.256} C_VEL
LIN {X 0,Y 599.977,Z 261.748,A -85,B 0,C 180,E1 112.092,E2 112.092} C_VEL
LIN {X 0,Y 599.922,Z 261.751,A -85,B 0,C 180,E1 108.966,E2 108.966} C_VEL
LIN {X 0,Y 599.972,Z 261.753,A -85,B 0,C 180,E1 105.862,E2 105.862} C_VEL
LIN {X 0,Y 599.911,Z 261.752,A -85,B 0,C 180,E1 102.834,E2 102.834} C_VEL
LIN {X 0,Y 599.922,Z 261.755,A -85,B 0,C 180,E1 99.595,E2 99.595} C_VEL
LIN {X 0,Y 599.905,Z 261.757,A -85,B 0,C 180,E1 96.701,E2 96.701} C_VEL
LIN {X 0,Y 599.985,Z 262.18,A -85,B 0,C 180,E1 96.508,E2 96.508} C_VEL
LIN {X 0,Y 600.494,Z 265.704,A -85,B 0,C 180,E1 96.214,E2 96.214} C_VEL
LIN {X 0,Y 600.557,Z 294.621,A -85,B 0,C 180,E1 94.011,E2 94.011} C_VEL
LIN {X 0,Y 600.422,Z 335.458,A -85,B 0,C 180,E1 90.907,E2 90.907} C_VEL
LIN {X 0,Y 600.294,Z 376.693,A -85,B 0,C 180,E1 87.853,E2 87.853} C_VEL
LIN {X 0,Y 600.211,Z 418.923,A -85,B 0,C 180,E1 84.792,E2 84.792} C_VEL
LIN {X 0,Y 600.106,Z 464.253,A -85,B 0,C 180,E1 81.57,E2 81.57} C_VEL
LIN {X 0,Y 600.166,Z 472.786,A -85,B 0,C 180,E1 81.001,E2 81.001} C_VEL
LIN {X 0,Y 600.135,Z 615.243,A -85,B 0,C 180,E1 79.241,E2 79.241} C_VEL
LIN {X 0,Y 600.133,Z 632.155,A -85,B 0,C 180,E1 78.84,E2 78.84} C_VEL
LIN {X 0,Y 600.099,Z 646.835,A -85,B 0,C 180,E1 78.322,E2 78.322} C_VEL
LIN {X 0,Y 600.061,Z 662.094,A -85,B 0,C 180,E1 77.589,E2 77.589} C_VEL
LIN {X 0,Y 600.029,Z 676.504,A -85,B 0,C 180,E1 76.695,E2 76.695} C_VEL
LIN {X 0,Y 599.994,Z 689.443,A -85,B 0,C 180,E1 75.674,E2 75.674} C_VEL
LIN {X 0,Y 599.968,Z 701.086,A -85,B 0,C 180,E1 74.537,E2 74.537} C_VEL
LIN {X 0,Y 599.945,Z 711.629,A -85,B 0,C 180,E1 73.244,E2 73.244} C_VEL
LIN {X 0,Y 599.933,Z 720.689,A -85,B 0,C 180,E1 71.842,E2 71.842} C_VEL
LIN {X 0,Y 599.919,Z 727.663,A -85,B 0,C 180,E1 70.429,E2 70.429} C_VEL
LIN {X 0,Y 599.915,Z 733.208,A -85,B 0,C 180,E1 68.901,E2 68.901} C_VEL
LIN {X 0,Y 599.914,Z 736.863,A -85,B 0,C 180,E1 67.358,E2 67.358} C_VEL
LIN {X 0,Y 599.916,Z 738.786,A -85,B 0,C 180,E1 65.692,E2 65.692} C_VEL
LIN {X 0,Y 599.914,Z 738.746,A -85,B 0,C 180,E1 64.16,E2 64.16} C_VEL
LIN {X 0,Y 599.915,Z 736.787,A -85,B 0,C 180,E1 62.507,E2 62.507} C_VEL
LIN {X 0,Y 599.915,Z 733.146,A -85,B 0,C 180,E1 60.989,E2 60.989} C_VEL
LIN {X 0,Y 599.922,Z 727.529,A -85,B 0,C 180,E1 59.449,E2 59.449} C_VEL
LIN {X 0,Y 599.931,Z 720.468,A -85,B 0,C 180,E1 58.029,E2 58.029} C_VEL
LIN {X 0,Y 599.944,Z 711.414,A -85,B 0,C 180,E1 56.637,E2 56.637} C_VEL
LIN {X 0,Y 599.969,Z 701.066,A -85,B 0,C 180,E1 55.371,E2 55.371} C_VEL
LIN {X 0,Y 599.994,Z 689.078,A -85,B 0,C 180,E1 54.204,E2 54.204} C_VEL
LIN {X 0,Y 600.031,Z 676.113,A -85,B 0,C 180,E1 53.189,E2 53.189} C_VEL
LIN {X 0,Y 600.058,Z 661.752,A -85,B 0,C 180,E1 52.302,E2 52.302} C_VEL
LIN {X 0,Y 600.086,Z 647.798,A -85,B 0,C 180,E1 51.629,E2 51.629} C_VEL
LIN {X 0,Y 600.132,Z 632.099,A -85,B 0,C 180,E1 51.069,E2 51.069} C_VEL
LIN {X 0,Y 600.123,Z 615.12,A -85,B 0,C 180,E1 50.667,E2 50.667} C_VEL
LIN {X 0,Y 600.114,Z 472.239,A -85,B 0,C 180,E1 48.893,E2 48.893} C_VEL
LIN {X 0,Y 600.13,Z 431.749,A -85,B 0,C 180,E1 46.034,E2 46.034} C_VEL
LIN {X 0,Y 600.243,Z 387.092,A -85,B 0,C 180,E1 42.815,E2 42.815} C_VEL
LIN {X 0,Y 600.39,Z 347.187,A -85,B 0,C 180,E1 39.879,E2 39.879} C_VEL
LIN {X 0,Y 600.534,Z 305.133,A -85,B 0,C 180,E1 36.707,E2 36.707} C_VEL
LIN {X 0,Y 600.531,Z 270.72,A -85,B 0,C 180,E1 34.074,E2 34.074} C_VEL
LIN {X 0,Y 600.134,Z 262.619,A -85,B 0,C 180,E1 33.468,E2 33.468} C_VEL
LIN {X 0,Y 599.97,Z 261.765,A -85,B 0,C 180,E1 33.291,E2 33.291} C_VEL
LIN {X 0,Y 599.935,Z 261.753,A -85,B 0,C 180,E1 30.22,E2 30.22} C_VEL
LIN {X 0,Y 599.94,Z 261.748,A -85,B 0,C 180,E1 26.925,E2 26.925} C_VEL
LIN {X 0,Y 599.972,Z 261.754,A -85,B 0,C 180,E1 23.785,E2 23.785} C_VEL
LIN {X 0,Y 599.929,Z 261.749,A -85,B 0,C 180,E1 20.589,E2 20.589} C_VEL
LIN {X 0,Y 599.976,Z 261.75,A -85,B 0,C 180,E1 17.456,E2 17.456} C_VEL
LIN {X 0,Y 599.928,Z 261.75,A -85,B 0,C 180,E1 14.379,E2 14.379} C_VEL
LIN {X 0,Y 599.975,Z 261.747,A -85,B 0,C 180,E1 11.244,E2 11.244} C_VEL
LIN {X 0,Y 599.933,Z 261.751,A -85,B 0,C 180,E1 8.135,E2 8.135} C_VEL
LIN {X 0,Y 599.959,Z 261.746,A -85,B 0,C 180,E1 4.876,E2 4.876} C_VEL
LIN {X 0,Y 599.959,Z 261.753,A -85,B 0,C 180,E1 1.719,E2 1.719} C_VEL
LIN {X 0,Y 599.935,Z 261.748,A -85,B 0,C 180,E1 -1.528,E2 -1.528} C_VEL
LIN {X 0,Y 599.975,Z 261.751,A -85,B 0,C 180,E1 -4.684,E2 -4.684} C_VEL
LIN {X 0,Y 599.931,Z 261.75,A -85,B 0,C 180,E1 -7.854,E2 -7.854} C_VEL
LIN {X 0,Y 599.976,Z 261.746,A -85,B 0,C 180,E1 -11.049,E2 -11.049} C_VEL
LIN {X 0,Y 599.942,Z 261.751,A -85,B 0,C 180,E1 -14.181,E2 -14.181} C_VEL
LIN {X 0,Y 599.952,Z 261.746,A -85,B 0,C 180,E1 -17.456,E2 -17.456} C_VEL
LIN {X 0,Y 599.978,Z 261.753,A -85,B 0,C 180,E1 -20.689,E2 -20.689} C_VEL
LIN {X 0,Y 599.935,Z 261.749,A -85,B 0,C 180,E1 -23.89,E2 -23.89} C_VEL
LIN {X 0,Y 599.973,Z 261.748,A -85,B 0,C 180,E1 -27.062,E2 -27.062} C_VEL
LIN {X 0,Y 599.94,Z 261.75,A -85,B 0,C 180,E1 -30.219,E2 -30.219} C_VEL
LIN {X 0,Y 599.969,Z 261.745,A -85,B 0,C 180,E1 -33.478,E2 -33.478} C_VEL
LIN {X 0,Y 599.975,Z 261.754,A -85,B 0,C 180,E1 -36.746,E2 -36.746} C_VEL
LIN {X 0,Y 599.94,Z 261.748,A -85,B 0,C 180,E1 -39.95,E2 -39.95} C_VEL
LIN {X 0,Y 599.972,Z 261.75,A -85,B 0,C 180,E1 -43.099,E2 -43.099} C_VEL
LIN {X 0,Y 599.939,Z 261.749,A -85,B 0,C 180,E1 -46.242,E2 -46.242} C_VEL
LIN {X 0,Y 599.974,Z 261.746,A -85,B 0,C 180,E1 -49.465,E2 -49.465} C_VEL
LIN {X 0,Y 599.954,Z 261.753,A -85,B 0,C 180,E1 -52.656,E2 -52.656} C_VEL
LIN {X 0,Y 599.951,Z 261.748,A -85,B 0,C 180,E1 -55.948,E2 -55.948} C_VEL
LIN {X 0,Y 599.976,Z 261.995,A -85,B 0,C 180,E1 -58.411,E2 -58.411} C_VEL
LIN {X 0,Y 600.75,Z 265.362,A -85,B 0,C 180,E1 -58.718,E2 -58.718} C_VEL
LIN {X 0,Y 600.583,Z 311.765,A -85,B 0,C 180,E1 -61.725,E2 -61.725} C_VEL
LIN {X 0,Y 600.704,Z 316.046,A -85,B 0,C 180,E1 -61.962,E2 -61.962} C_VEL
LIN {X 0,Y 600.667,Z 519.783,A -85,B 0,C 180,E1 -64.633,E2 -64.633} C_VEL
LIN {X 0,Y 600.61,Z 578.292,A -85,B 0,C 180,E1 -65.417,E2 -65.417} C_VEL
LIN {X 0,Y 600.557,Z 598.764,A -85,B 0,C 180,E1 -65.876,E2 -65.876} C_VEL
LIN {X 0,Y 600.499,Z 617.817,A -85,B 0,C 180,E1 -66.474,E2 -66.474} C_VEL
LIN {X 0,Y 600.425,Z 637.639,A -85,B 0,C 180,E1 -67.275,E2 -67.275} C_VEL
LIN {X 0,Y 600.349,Z 656.078,A -85,B 0,C 180,E1 -68.2,E2 -68.2} C_VEL
LIN {X 0,Y 600.277,Z 674.551,A -85,B 0,C 180,E1 -69.323,E2 -69.323} C_VEL
LIN {X 0,Y 600.197,Z 692.585,A -85,B 0,C 180,E1 -70.641,E2 -70.641} C_VEL
LIN {X 0,Y 600.123,Z 709.379,A -85,B 0,C 180,E1 -72.099,E2 -72.099} C_VEL
LIN {X 0,Y 600.064,Z 724.878,A -85,B 0,C 180,E1 -73.691,E2 -73.691} C_VEL
LIN {X 0,Y 600.007,Z 738.373,A -85,B 0,C 180,E1 -75.329,E2 -75.329} C_VEL
LIN {X 0,Y 599.972,Z 750.023,A -85,B 0,C 180,E1 -77,E2 -77} C_VEL
LIN {X 0,Y 599.945,Z 760.331,A -85,B 0,C 180,E1 -78.757,E2 -78.757} C_VEL
LIN {X 0,Y 599.925,Z 769.36,A -85,B 0,C 180,E1 -80.627,E2 -80.627} C_VEL
LIN {X 0,Y 599.92,Z 776.383,A -85,B 0,C 180,E1 -82.435,E2 -82.435} C_VEL
LIN {X 0,Y 599.913,Z 782.004,A -85,B 0,C 180,E1 -84.358,E2 -84.358} C_VEL
LIN {X 0,Y 599.912,Z 785.926,A -85,B 0,C 180,E1 -86.274,E2 -86.274} C_VEL
LIN {X 0,Y 599.906,Z 788.307,A -85,B 0,C 180,E1 -88.282,E2 -88.282} C_VEL
LIN {X 0,Y 599.907,Z 788.962,A -85,B 0,C 180,E1 -90.192,E2 -90.192} C_VEL
LIN {X 0,Y 599.91,Z 787.949,A -85,B 0,C 180,E1 -92.198,E2 -92.198} C_VEL
LIN {X 0,Y 599.909,Z 785.133,A -85,B 0,C 180,E1 -94.206,E2 -94.206} C_VEL
LIN {X 0,Y 599.919,Z 780.733,A -85,B 0,C 180,E1 -96.124,E2 -96.124} C_VEL
LIN {X 0,Y 599.923,Z 774.616,A -85,B 0,C 180,E1 -98.049,E2 -98.049} C_VEL
LIN {X 0,Y 599.934,Z 766.799,A -85,B 0,C 180,E1 -99.947,E2 -99.947} C_VEL
LIN {X 0,Y 599.943,Z 757.711,A -85,B 0,C 180,E1 -101.732,E2 -101.732} C_VEL
LIN {X 0,Y 599.974,Z 746.81,A -85,B 0,C 180,E1 -103.493,E2 -103.493} C_VEL
LIN {X 0,Y 600.019,Z 734.479,A -85,B 0,C 180,E1 -105.167,E2 -105.167} C_VEL
LIN {X 0,Y 600.065,Z 720.733,A -85,B 0,C 180,E1 -106.755,E2 -106.755} C_VEL
LIN {X 0,Y 600.133,Z 705.441,A -85,B 0,C 180,E1 -108.259,E2 -108.259} C_VEL
LIN {X 0,Y 600.207,Z 688.595,A -85,B 0,C 180,E1 -109.665,E2 -109.665} C_VEL
LIN {X 0,Y 600.29,Z 671.337,A -85,B 0,C 180,E1 -110.883,E2 -110.883} C_VEL
LIN {X 0,Y 600.374,Z 653.234,A -85,B 0,C 180,E1 -111.956,E2 -111.956} C_VEL
LIN {X 0,Y 600.442,Z 634.219,A -85,B 0,C 180,E1 -112.882,E2 -112.882} C_VEL
LIN {X 0,Y 600.507,Z 614.815,A -85,B 0,C 180,E1 -113.632,E2 -113.632} C_VEL
LIN {X 0,Y 600.564,Z 594.781,A -85,B 0,C 180,E1 -114.224,E2 -114.224} C_VEL
LIN {X 0,Y 600.619,Z 574.279,A -85,B 0,C 180,E1 -114.646,E2 -114.646} C_VEL
LIN {X 0,Y 600.788,Z 328.828,A -85,B 0,C 180,E1 -117.863,E2 -117.863} C_VEL
LIN {X 0,Y 600.615,Z 315.45,A -85,B 0,C 180,E1 -118.054,E2 -118.054} C_VEL
LIN {X 0,Y 600.741,Z 269.622,A -85,B 0,C 180,E1 -121.002,E2 -121.002} C_VEL
LIN {X 0,Y 600.68,Z 264.235,A -85,B 0,C 180,E1 -121.361,E2 -121.361} C_VEL
LIN {X 0,Y 599.96,Z 261.887,A -85,B 0,C 180,E1 -121.614,E2 -121.614} C_VEL
LIN {X 0,Y 599.971,Z 261.752,A -85,B 0,C 180,E1 -124.756,E2 -124.756} C_VEL
LIN {X 0,Y 599.936,Z 261.749,A -85,B 0,C 180,E1 -127.83,E2 -127.83} C_VEL
LIN {X 0,Y 599.977,Z 261.754,A -85,B 0,C 180,E1 -131.042,E2 -131.042} C_VEL
LIN {X 0,Y 599.952,Z 261.747,A -85,B 0,C 180,E1 -134.224,E2 -134.224} C_VEL
LIN {X 0,Y 599.94,Z 261.752,A -85,B 0,C 180,E1 -137.446,E2 -137.446} C_VEL
LIN {X 0,Y 599.979,Z 261.747,A -85,B 0,C 180,E1 -140.585,E2 -140.585} C_VEL
LIN {X 0,Y 599.925,Z 261.751,A -85,B 0,C 180,E1 -143.771,E2 -143.771} C_VEL
LIN {X 0,Y 599.976,Z 261.752,A -85,B 0,C 180,E1 -146.865,E2 -146.865} C_VEL
LIN {X 0,Y 599.919,Z 261.744,A -85,B 0,C 180,E1 -149.89,E2 -149.89} C_VEL
LIN {X 0,Y 600.003,Z 262.027,A -85,B 0,C 180,E1 -150.57,E2 -150.57} C_VEL
LIN {X 0,Y 600.581,Z 265.108,A -85,B 0,C 180,E1 -150.859,E2 -150.859} C_VEL
LIN {X 0,Y 600.412,Z 305.124,A -85,B 0,C 180,E1 -153.844,E2 -153.844} C_VEL
LIN {X 0,Y 600.434,Z 342.643,A -85,B 0,C 180,E1 -156.55,E2 -156.55} C_VEL
LIN {X 0,Y 600.428,Z 548.25,A -85,B 0,C 180,E1 -159.157,E2 -159.157} C_VEL
LIN {X 0,Y 600.396,Z 568.16,A -85,B 0,C 180,E1 -159.489,E2 -159.489} C_VEL
LIN {X 0,Y 600.352,Z 587.649,A -85,B 0,C 180,E1 -160.006,E2 -160.006} C_VEL
LIN {X 0,Y 600.302,Z 605.96,A -85,B 0,C 180,E1 -160.676,E2 -160.676} C_VEL
LIN {X 0,Y 600.238,Z 623.416,A -85,B 0,C 180,E1 -161.499,E2 -161.499} C_VEL
LIN {X 0,Y 600.182,Z 640.833,A -85,B 0,C 180,E1 -162.518,E2 -162.518} C_VEL
LIN {X 0,Y 600.119,Z 657.022,A -85,B 0,C 180,E1 -163.674,E2 -163.674} C_VEL
LIN {X 0,Y 600.056,Z 672.23,A -85,B 0,C 180,E1 -164.983,E2 -164.983} C_VEL
LIN {X 0,Y 600.01,Z 686.053,A -85,B 0,C 180,E1 -166.411,E2 -166.411} C_VEL
LIN {X 0,Y 599.971,Z 697.976,A -85,B 0,C 180,E1 -167.879,E2 -167.879} C_VEL
LIN {X 0,Y 599.948,Z 708.519,A -85,B 0,C 180,E1 -169.437,E2 -169.437} C_VEL
LIN {X 0,Y 599.93,Z 717.663,A -85,B 0,C 180,E1 -171.084,E2 -171.084} C_VEL
LIN {X 0,Y 599.921,Z 725.343,A -85,B 0,C 180,E1 -172.82,E2 -172.82} C_VEL
LIN {X 0,Y 599.916,Z 731.456,A -85,B 0,C 180,E1 -174.645,E2 -174.645} C_VEL
LIN {X 0,Y 599.905,Z 735.71,A -85,B 0,C 180,E1 -176.465,E2 -176.465} C_VEL
LIN {X 0,Y 599.908,Z 738.196,A -85,B 0,C 180,E1 -178.281,E2 -178.281} C_VEL
LIN {X 0,Y 599.916,Z 738.994,A -85,B 0,C 180,E1 -180.096,E2 -180.096} C_VEL
LIN {X 0,Y 599.905,Z 738.107,A -85,B 0,C 180,E1 -181.911,E2 -181.911} C_VEL
LIN {X 0,Y 599.906,Z 735.523,A -85,B 0,C 180,E1 -183.727,E2 -183.727} C_VEL
LIN {X 0,Y 599.915,Z 731.175,A -85,B 0,C 180,E1 -185.548,E2 -185.548} C_VEL
LIN {X 0,Y 599.918,Z 728.211,A -85,B 0,C 180,E1 -186.486,E2 -186.486} C_VEL
LIN {X 0,Y 598.938,Z 725.736,A -85,B 0,C 180,E1 -187.183,E2 -187.183} C_VEL
LIN {X 0,Y 593.523,Z 719.553,A -85,B 0,C 180,E1 -188.715,E2 -188.715} C_VEL
LIN {X 0,Y 592.055,Z 716.348,A -85,B 0,C 180,E1 -189.388,E2 -189.388} C_VEL
LIN {X 0,Y 591.958,Z 715.339,A -85,B 0,C 180,E1 -189.581,E2 -189.581} C_VEL
LIN {X 0,Y 592.005,Z 705.364,A -85,B 0,C 180,E1 -191.299,E2 -191.299} C_VEL
LIN {X 0,Y 592.062,Z 694.15,A -85,B 0,C 180,E1 -192.881,E2 -192.881} C_VEL
LIN {X 0,Y 592.143,Z 681.452,A -85,B 0,C 180,E1 -194.372,E2 -194.372} C_VEL
LIN {X 0,Y 592.239,Z 667.137,A -85,B 0,C 180,E1 -195.779,E2 -195.779} C_VEL
LIN {X 0,Y 592.355,Z 651.963,A -85,B 0,C 180,E1 -197.024,E2 -197.024} C_VEL
LIN {X 0,Y 592.48,Z 635.562,A -85,B 0,C 180,E1 -198.142,E2 -198.142} C_VEL
LIN {X 0,Y 592.607,Z 617.997,A -85,B 0,C 180,E1 -199.118,E2 -199.118} C_VEL
LIN {X 0,Y 592.718,Z 601,A -85,B 0,C 180,E1 -199.872,E2 -199.872} C_VEL
LIN {X 0,Y 592.828,Z 582.281,A -85,B 0,C 180,E1 -200.512,E2 -200.512} C_VEL
LIN {X 0,Y 592.904,Z 563.275,A -85,B 0,C 180,E1 -200.971,E2 -200.971} C_VEL
LIN {X 0,Y 592.969,Z 536.355,A -85,B 0,C 180,E1 -201.36,E2 -201.36} C_VEL
LIN {X 0,Y 593.065,Z 343.72,A -85,B 0,C 180,E1 -203.831,E2 -203.831} C_VEL
LIN {X 0,Y 592.812,Z 341.522,A -85,B 0,C 180,E1 -203.913,E2 -203.913} C_VEL
LIN {X 0,Y 593.02,Z 299.426,A -85,B 0,C 180,E1 -207.026,E2 -207.026} C_VEL
LIN {X 0,Y 593.26,Z 266.996,A -85,B 0,C 180,E1 -209.481,E2 -209.481} C_VEL
LIN {X 0,Y 592.003,Z 262.881,A -85,B 0,C 180,E1 -209.912,E2 -209.912} C_VEL
LIN {X 0,Y 592.031,Z 262.736,A -85,B 0,C 180,E1 -212.944,E2 -212.944} C_VEL
LIN {X 0,Y 591.991,Z 262.739,A -85,B 0,C 180,E1 -216.119,E2 -216.119} C_VEL
LIN {X 0,Y 592.037,Z 262.736,A -85,B 0,C 180,E1 -219.296,E2 -219.296} C_VEL
LIN {X 0,Y 592.022,Z 262.741,A -85,B 0,C 180,E1 -222.577,E2 -222.577} C_VEL
LIN {X 0,Y 592.016,Z 262.736,A -85,B 0,C 180,E1 -225.873,E2 -225.873} C_VEL
LIN {X 0,Y 592.024,Z 262.738,A -85,B 0,C 180,E1 -229.058,E2 -229.058} C_VEL
LIN {X 0,Y 592.021,Z 262.739,A -85,B 0,C 180,E1 -232.224,E2 -232.224} C_VEL
LIN {X 0,Y 592.025,Z 262.734,A -85,B 0,C 180,E1 -235.426,E2 -235.426} C_VEL
LIN {X 0,Y 592.015,Z 262.74,A -85,B 0,C 180,E1 -238.768,E2 -238.768} C_VEL
LIN {X 0,Y 592.033,Z 262.737,A -85,B 0,C 180,E1 -241.997,E2 -241.997} C_VEL
LIN {X 0,Y 591.998,Z 262.737,A -85,B 0,C 180,E1 -245.13,E2 -245.13} C_VEL
LIN {X 0,Y 592.032,Z 262.741,A -85,B 0,C 180,E1 -248.292,E2 -248.292} C_VEL
LIN {X 0,Y 592.006,Z 262.738,A -85,B 0,C 180,E1 -251.486,E2 -251.486} C_VEL
LIN {X 0,Y 591.979,Z 262.739,A -85,B 0,C 180,E1 -254.722,E2 -254.722} C_VEL
LIN {X 0,Y 592.028,Z 262.74,A -85,B 0,C 180,E1 -257.812,E2 -257.812} C_VEL
LIN {X 0,Y 591.958,Z 262.745,A -85,B 0,C 180,E1 -260.863,E2 -260.863} C_VEL
LIN {X 0,Y 591.993,Z 262.99,A -85,B 0,C 180,E1 -263.173,E2 -263.173} C_VEL
LIN {X 0,Y 593.004,Z 267.28,A -85,B 0,C 180,E1 -263.561,E2 -263.561} C_VEL
LIN {X 0,Y 593.163,Z 305.254,A -85,B 0,C 180,E1 -266.423,E2 -266.423} C_VEL
LIN {X 0,Y 592.909,Z 347.591,A -85,B 0,C 180,E1 -269.661,E2 -269.661} C_VEL
LIN {X 0,Y 592.643,Z 388.451,A -85,B 0,C 180,E1 -272.707,E2 -272.707} C_VEL
LIN {X 0,Y 592.468,Z 432.944,A -85,B 0,C 180,E1 -275.956,E2 -275.956} C_VEL
LIN {X 0,Y 592.369,Z 472.692,A -85,B 0,C 180,E1 -278.781,E2 -278.781} C_VEL
LIN {X 0,Y 592.377,Z 615.341,A -85,B 0,C 180,E1 -280.57,E2 -280.57} C_VEL
LIN {X 0,Y 592.353,Z 632.233,A -85,B 0,C 180,E1 -280.976,E2 -280.976} C_VEL
LIN {X 0,Y 592.279,Z 648.091,A -85,B 0,C 180,E1 -281.553,E2 -281.553} C_VEL
LIN {X 0,Y 592.206,Z 663.716,A -85,B 0,C 180,E1 -282.331,E2 -282.331} C_VEL
LIN {X 0,Y 592.135,Z 677.581,A -85,B 0,C 180,E1 -283.225,E2 -283.225} C_VEL
LIN {X 0,Y 592.069,Z 691.026,A -85,B 0,C 180,E1 -284.323,E2 -284.323} C_VEL
LIN {X 0,Y 592.013,Z 702.334,A -85,B 0,C 180,E1 -285.476,E2 -285.476} C_VEL
LIN {X 0,Y 591.971,Z 712.659,A -85,B 0,C 180,E1 -286.786,E2 -286.786} C_VEL
LIN {X 0,Y 591.946,Z 720.917,A -85,B 0,C 180,E1 -288.106,E2 -288.106} C_VEL
LIN {X 0,Y 591.924,Z 727.836,A -85,B 0,C 180,E1 -289.538,E2 -289.538} C_VEL
LIN {X 0,Y 591.917,Z 733.333,A -85,B 0,C 180,E1 -291.086,E2 -291.086} C_VEL
LIN {X 0,Y 591.914,Z 736.929,A -85,B 0,C 180,E1 -292.651,E2 -292.651} C_VEL
LIN {X 0,Y 591.917,Z 738.742,A -85,B 0,C 180,E1 -294.233,E2 -294.233} C_VEL
LIN {X 0,Y 591.914,Z 738.784,A -85,B 0,C 180,E1 -295.796,E2 -295.796} C_VEL
LIN {X 0,Y 591.915,Z 736.894,A -85,B 0,C 180,E1 -297.46,E2 -297.46} C_VEL
LIN {X 0,Y 591.917,Z 733.353,A -85,B 0,C 180,E1 -298.998,E2 -298.998} C_VEL
LIN {X 0,Y 591.927,Z 727.81,A -85,B 0,C 180,E1 -300.558,E2 -300.558} C_VEL
LIN {X 0,Y 591.946,Z 720.667,A -85,B 0,C 180,E1 -302.029,E2 -302.029} C_VEL
LIN {X 0,Y 591.974,Z 711.62,A -85,B 0,C 180,E1 -303.448,E2 -303.448} C_VEL
LIN {X 0,Y 592.019,Z 701.684,A -85,B 0,C 180,E1 -304.69,E2 -304.69} C_VEL
LIN {X 0,Y 592.072,Z 689.863,A -85,B 0,C 180,E1 -305.871,E2 -305.871} C_VEL
LIN {X 0,Y 592.138,Z 677.349,A -85,B 0,C 180,E1 -306.882,E2 -306.882} C_VEL
LIN {X 0,Y 592.203,Z 663.732,A -85,B 0,C 180,E1 -307.758,E2 -307.758} C_VEL
LIN {X 0,Y 592.271,Z 648.277,A -85,B 0,C 180,E1 -308.529,E2 -308.529} C_VEL
LIN {X 0,Y 592.352,Z 632.347,A -85,B 0,C 180,E1 -309.11,E2 -309.11} C_VEL
LIN {X 0,Y 592.365,Z 615.505,A -85,B 0,C 180,E1 -309.518,E2 -309.518} C_VEL
LIN {X 0,Y 592.453,Z 528.737,A -85,B 0,C 180,E1 -310.609,E2 -310.609} C_VEL
LIN {X 0,Y 592.327,Z 472.394,A -85,B 0,C 180,E1 -311.317,E2 -311.317} C_VEL
LIN {X 0,Y 592.424,Z 432.221,A -85,B 0,C 180,E1 -314.188,E2 -314.188} C_VEL
LIN {X 0,Y 592.635,Z 386.909,A -85,B 0,C 180,E1 -317.498,E2 -317.498} C_VEL
LIN {X 0,Y 592.897,Z 347.818,A -85,B 0,C 180,E1 -320.413,E2 -320.413} C_VEL
LIN {X 0,Y 593.165,Z 306.048,A -85,B 0,C 180,E1 -323.605,E2 -323.605} C_VEL
LIN {X 0,Y 592.968,Z 269.99,A -85,B 0,C 180,E1 -326.305,E2 -326.305} C_VEL
LIN {X 0,Y 592.591,Z 264.884,A -85,B 0,C 180,E1 -326.687,E2 -326.687} C_VEL
LIN {X 0,Y 592.038,Z 262.941,A -85,B 0,C 180,E1 -326.891,E2 -326.891} C_VEL
LIN {X 0,Y 592.004,Z 262.744,A -85,B 0,C 180,E1 -329.893,E2 -329.893} C_VEL
LIN {X 0,Y 591.995,Z 262.738,A -85,B 0,C 180,E1 -333.195,E2 -333.195} C_VEL
LIN {X 0,Y 592.038,Z 262.742,A -85,B 0,C 180,E1 -336.3,E2 -336.3} C_VEL
LIN {X 0,Y 591.989,Z 262.738,A -85,B 0,C 180,E1 -339.432,E2 -339.432} C_VEL
LIN {X 0,Y 592.037,Z 262.738,A -85,B 0,C 180,E1 -342.607,E2 -342.607} C_VEL
LIN {X 0,Y 591.994,Z 262.74,A -85,B 0,C 180,E1 -345.798,E2 -345.798} C_VEL
LIN {X 0,Y 592.017,Z 262.735,A -85,B 0,C 180,E1 -349.096,E2 -349.096} C_VEL
LIN {X 0,Y 592.032,Z 262.742,A -85,B 0,C 180,E1 -352.332,E2 -352.332} C_VEL
LIN {X 0,Y 591.993,Z 262.738,A -85,B 0,C 180,E1 -355.544,E2 -355.544} C_VEL
LIN {X 0,Y 592.037,Z 262.738,A -85,B 0,C 180,E1 -358.742,E2 -358.742} C_VEL
LIN {X 0,Y 591.993,Z 262.739,A -85,B 0,C 180,E1 -361.839,E2 -361.839} C_VEL
LIN {X 0,Y 592.037,Z 262.735,A -85,B 0,C 180,E1 -365.038,E2 -365.038} C_VEL
LIN {X 0,Y 592.009,Z 262.741,A -85,B 0,C 180,E1 -368.253,E2 -368.253} C_VEL
LIN {X 0,Y 592.006,Z 262.736,A -85,B 0,C 180,E1 -371.495,E2 -371.495} C_VEL
LIN {X 0,Y 592.039,Z 262.741,A -85,B 0,C 180,E1 -374.674,E2 -374.674} C_VEL
LIN {X 0,Y 591.995,Z 262.738,A -85,B 0,C 180,E1 -377.902,E2 -377.902} C_VEL
LIN {X 0,Y 592.037,Z 262.735,A -85,B 0,C 180,E1 -381.083,E2 -381.083} C_VEL
LIN {X 0,Y 592.003,Z 262.74,A -85,B 0,C 180,E1 -384.23,E2 -384.23} C_VEL
LIN {X 0,Y 592.014,Z 262.735,A -85,B 0,C 180,E1 -387.565,E2 -387.565} C_VEL
LIN {X 0,Y 592.04,Z 262.742,A -85,B 0,C 180,E1 -390.778,E2 -390.778} C_VEL
LIN {X 0,Y 591.999,Z 262.737,A -85,B 0,C 180,E1 -393.989,E2 -393.989} C_VEL
LIN {X 0,Y 592.034,Z 262.737,A -85,B 0,C 180,E1 -397.145,E2 -397.145} C_VEL
LIN {X 0,Y 592.002,Z 262.739,A -85,B 0,C 180,E1 -400.305,E2 -400.305} C_VEL
LIN {X 0,Y 592.03,Z 262.734,A -85,B 0,C 180,E1 -403.573,E2 -403.573} C_VEL
LIN {X 0,Y 592.037,Z 262.743,A -85,B 0,C 180,E1 -406.851,E2 -406.851} C_VEL
LIN {X 0,Y 592.002,Z 262.737,A -85,B 0,C 180,E1 -410.076,E2 -410.076} C_VEL
LIN {X 0,Y 592.031,Z 262.732,A -85,B 0,C 180,E1 -413.179,E2 -413.179} C_VEL
LIN {X 0,Y 592.003,Z 262.742,A -85,B 0,C 180,E1 -416.371,E2 -416.371} C_VEL
LIN {X 0,Y 592.046,Z 262.985,A -85,B 0,C 180,E1 -418.005,E2 -418.005} C_VEL
LIN {X 0,Y 593.599,Z 267.831,A -85,B 0,C 180,E1 -418.463,E2 -418.463} C_VEL
LIN {X 0,Y 593.279,Z 314.401,A -85,B 0,C 180,E1 -421.516,E2 -421.516} C_VEL
LIN {X 0,Y 593.728,Z 318.555,A -85,B 0,C 180,E1 -421.638,E2 -421.638} C_VEL
LIN {X 0,Y 593.386,Z 547.087,A -85,B 0,C 180,E1 -424.658,E2 -424.658} C_VEL
LIN {X 0,Y 593.313,Z 579.752,A -85,B 0,C 180,E1 -425.125,E2 -425.125} C_VEL
LIN {X 0,Y 593.22,Z 600.256,A -85,B 0,C 180,E1 -425.597,E2 -425.597} C_VEL
LIN {X 0,Y 593.093,Z 620.024,A -85,B 0,C 180,E1 -426.241,E2 -426.241} C_VEL
LIN {X 0,Y 592.946,Z 638.839,A -85,B 0,C 180,E1 -427.028,E2 -427.028} C_VEL
LIN {X 0,Y 592.782,Z 657.865,A -85,B 0,C 180,E1 -428.011,E2 -428.011} C_VEL
LIN {X 0,Y 592.626,Z 676.018,A -85,B 0,C 180,E1 -429.147,E2 -429.147} C_VEL
LIN {X 0,Y 592.481,Z 693.207,A -85,B 0,C 180,E1 -430.43,E2 -430.43} C_VEL
LIN {X 0,Y 592.335,Z 709.911,A -85,B 0,C 180,E1 -431.907,E2 -431.907} C_VEL
LIN {X 0,Y 592.21,Z 725.363,A -85,B 0,C 180,E1 -433.524,E2 -433.524} C_VEL
LIN {X 0,Y 592.103,Z 739.141,A -85,B 0,C 180,E1 -435.228,E2 -435.228} C_VEL
LIN {X 0,Y 592.03,Z 751.335,A -85,B 0,C 180,E1 -437.026,E2 -437.026} C_VEL
LIN {X 0,Y 591.975,Z 761.369,A -85,B 0,C 180,E1 -438.801,E2 -438.801} C_VEL
LIN {X 0,Y 591.936,Z 770.066,A -85,B 0,C 180,E1 -440.669,E2 -440.669} C_VEL
LIN {X 0,Y 591.917,Z 777.052,A -85,B 0,C 180,E1 -442.546,E2 -442.546} C_VEL
LIN {X 0,Y 591.909,Z 782.51,A -85,B 0,C 180,E1 -444.476,E2 -444.476} C_VEL
LIN {X 0,Y 591.904,Z 786.242,A -85,B 0,C 180,E1 -446.418,E2 -446.418} C_VEL
LIN {X 0,Y 591.903,Z 788.374,A -85,B 0,C 180,E1 -448.355,E2 -448.355} C_VEL
LIN {X 0,Y 591.9,Z 788.917,A -85,B 0,C 180,E1 -450.388,E2 -450.388} C_VEL
LIN {X 0,Y 591.905,Z 787.838,A -85,B 0,C 180,E1 -452.325,E2 -452.325} C_VEL
LIN {X 0,Y 591.908,Z 784.971,A -85,B 0,C 180,E1 -454.361,E2 -454.361} C_VEL
LIN {X 0,Y 591.918,Z 780.48,A -85,B 0,C 180,E1 -456.305,E2 -456.305} C_VEL
LIN {X 0,Y 591.934,Z 774.262,A -85,B 0,C 180,E1 -458.256,E2 -458.256} C_VEL
LIN {X 0,Y 591.96,Z 766.172,A -85,B 0,C 180,E1 -460.216,E2 -460.216} C_VEL
LIN {X 0,Y 592.001,Z 756.562,A -85,B 0,C 180,E1 -462.09,E2 -462.09} C_VEL
LIN {X 0,Y 592.068,Z 745.492,A -85,B 0,C 180,E1 -463.876,E2 -463.876} C_VEL
LIN {X 0,Y 592.143,Z 732.929,A -85,B 0,C 180,E1 -465.575,E2 -465.575} C_VEL
LIN {X 0,Y 592.249,Z 718.879,A -85,B 0,C 180,E1 -467.185,E2 -467.185} C_VEL
LIN {X 0,Y 592.37,Z 703.835,A -85,B 0,C 180,E1 -468.655,E2 -468.655} C_VEL
LIN {X 0,Y 592.518,Z 687.276,A -85,B 0,C 180,E1 -470.034,E2 -470.034} C_VEL
LIN {X 0,Y 592.682,Z 669.735,A -85,B 0,C 180,E1 -471.267,E2 -471.267} C_VEL
LIN {X 0,Y 592.85,Z 651.248,A -85,B 0,C 180,E1 -472.354,E2 -472.354} C_VEL
LIN {X 0,Y 593.009,Z 632.397,A -85,B 0,C 180,E1 -473.265,E2 -473.265} C_VEL
LIN {X 0,Y 593.136,Z 612.748,A -85,B 0,C 180,E1 -474.018,E2 -474.018} C_VEL
LIN {X 0,Y 593.246,Z 592.965,A -85,B 0,C 180,E1 -474.588,E2 -474.588} C_VEL
LIN {X 0,Y 593.342,Z 572.319,A -85,B 0,C 180,E1 -475,E2 -475} C_VEL
LIN {X 0,Y 593.712,Z 329.973,A -85,B 0,C 180,E1 -478.209,E2 -478.209} C_VEL
LIN {X 0,Y 593.498,Z 316.574,A -85,B 0,C 180,E1 -478.4,E2 -478.4} C_VEL
LIN {X 0,Y 593.277,Z 314.36,A -85,B 0,C 180,E1 -478.487,E2 -478.487} C_VEL
LIN {X 0,Y 593.6,Z 267.671,A -85,B 0,C 180,E1 -481.548,E2 -481.548} C_VEL
LIN {X 0,Y 592.041,Z 262.954,A -85,B 0,C 180,E1 -481.998,E2 -481.998} C_VEL
LIN {X 0,Y 592.027,Z 262.744,A -85,B 0,C 180,E1 -485.173,E2 -485.173} C_VEL
LIN {X 0,Y 592.039,Z 262.735,A -85,B 0,C 180,E1 -488.426,E2 -488.426} C_VEL
LIN {X 0,Y 591.998,Z 262.74,A -85,B 0,C 180,E1 -491.588,E2 -491.588} C_VEL
LIN {X 0,Y 592.036,Z 262.739,A -85,B 0,C 180,E1 -494.77,E2 -494.77} C_VEL
LIN {X 0,Y 591.991,Z 262.739,A -85,B 0,C 180,E1 -497.893,E2 -497.893} C_VEL
LIN {X 0,Y 592.028,Z 262.744,A -85,B 0,C 180,E1 -501.131,E2 -501.131} C_VEL
LIN {X 0,Y 592,Z 262.739,A -85,B 0,C 180,E1 -504.241,E2 -504.241} C_VEL
LIN {X 0,Y 591.994,Z 262.744,A -85,B 0,C 180,E1 -507.514,E2 -507.514} C_VEL
LIN {X 0,Y 592.025,Z 262.972,A -85,B 0,C 180,E1 -510.202,E2 -510.202} C_VEL
LIN {X 0,Y 593.256,Z 267.278,A -85,B 0,C 180,E1 -510.631,E2 -510.631} C_VEL
LIN {X 0,Y 592.959,Z 307.602,A -85,B 0,C 180,E1 -513.674,E2 -513.674} C_VEL
LIN {X 0,Y 592.881,Z 342.554,A -85,B 0,C 180,E1 -516.231,E2 -516.231} C_VEL
LIN {X 0,Y 593.208,Z 348.346,A -85,B 0,C 180,E1 -516.325,E2 -516.325} C_VEL
LIN {X 0,Y 592.919,Z 559.862,A -85,B 0,C 180,E1 -519.053,E2 -519.053} C_VEL
LIN {X 0,Y 592.841,Z 579.487,A -85,B 0,C 180,E1 -519.496,E2 -519.496} C_VEL
LIN {X 0,Y 592.742,Z 598.141,A -85,B 0,C 180,E1 -520.104,E2 -520.104} C_VEL
LIN {X 0,Y 592.625,Z 616.45,A -85,B 0,C 180,E1 -520.895,E2 -520.895} C_VEL
LIN {X 0,Y 592.5,Z 634.151,A -85,B 0,C 180,E1 -521.86,E2 -521.86} C_VEL
LIN {X 0,Y 592.37,Z 650.762,A -85,B 0,C 180,E1 -522.975,E2 -522.975} C_VEL
LIN {X 0,Y 592.25,Z 666.231,A -85,B 0,C 180,E1 -524.229,E2 -524.229} C_VEL
LIN {X 0,Y 592.145,Z 680.62,A -85,B 0,C 180,E1 -525.628,E2 -525.628} C_VEL
LIN {X 0,Y 592.064,Z 693.453,A -85,B 0,C 180,E1 -527.12,E2 -527.12} C_VEL
LIN {X 0,Y 592.008,Z 704.786,A -85,B 0,C 180,E1 -528.702,E2 -528.702} C_VEL
LIN {X 0,Y 591.957,Z 714.631,A -85,B 0,C 180,E1 -530.374,E2 -530.374} C_VEL
LIN {X 0,Y 591.933,Z 722.961,A -85,B 0,C 180,E1 -532.136,E2 -532.136} C_VEL
LIN {X 0,Y 591.913,Z 729.701,A -85,B 0,C 180,E1 -533.989,E2 -533.989} C_VEL
LIN {X 0,Y 591.91,Z 734.529,A -85,B 0,C 180,E1 -535.835,E2 -535.835} C_VEL
LIN {X 0,Y 591.914,Z 737.563,A -85,B 0,C 180,E1 -537.677,E2 -537.677} C_VEL
LIN {X 0,Y 591.905,Z 738.907,A -85,B 0,C 180,E1 -539.613,E2 -539.613} C_VEL
LIN {X 0,Y 591.912,Z 738.463,A -85,B 0,C 180,E1 -541.452,E2 -541.452} C_VEL
LIN {X 0,Y 591.915,Z 736.279,A -85,B 0,C 180,E1 -543.324,E2 -543.324} C_VEL
LIN {X 0,Y 591.919,Z 732.451,A -85,B 0,C 180,E1 -545.137,E2 -545.137} C_VEL
LIN {X 0,Y 591.926,Z 726.728,A -85,B 0,C 180,E1 -546.986,E2 -546.986} C_VEL
LIN {X 0,Y 591.947,Z 719.467,A -85,B 0,C 180,E1 -548.744,E2 -548.744} C_VEL
LIN {X 0,Y 591.958,Z 715.339,A -85,B 0,C 180,E1 -549.581,E2 -549.581} C_VEL
LIN {X 0,Y 590.959,Z 711.867,A -85,B 0,C 180,E1 -550.244,E2 -550.244} C_VEL
LIN {X 0,Y 585.038,Z 702.472,A -85,B 0,C 180,E1 -551.883,E2 -551.883} C_VEL
LIN {X 0,Y 584.108,Z 698.186,A -85,B 0,C 180,E1 -552.518,E2 -552.518} C_VEL
LIN {X 0,Y 584.224,Z 685.972,A -85,B 0,C 180,E1 -554.065,E2 -554.065} C_VEL
LIN {X 0,Y 584.365,Z 672.622,A -85,B 0,C 180,E1 -555.481,E2 -555.481} C_VEL
LIN {X 0,Y 584.538,Z 657.783,A -85,B 0,C 180,E1 -556.803,E2 -556.803} C_VEL
LIN {X 0,Y 584.724,Z 641.916,A -85,B 0,C 180,E1 -557.978,E2 -557.978} C_VEL
LIN {X 0,Y 584.918,Z 624.153,A -85,B 0,C 180,E1 -559.057,E2 -559.057} C_VEL
LIN {X 0,Y 585.112,Z 606.068,A -85,B 0,C 180,E1 -559.933,E2 -559.933} C_VEL
LIN {X 0,Y 585.274,Z 587.255,A -85,B 0,C 180,E1 -560.636,E2 -560.636} C_VEL
LIN {X 0,Y 585.408,Z 567.774,A -85,B 0,C 180,E1 -561.161,E2 -561.161} C_VEL
LIN {X 0,Y 585.497,Z 547.656,A -85,B 0,C 180,E1 -561.499,E2 -561.499} C_VEL
LIN {X 0,Y 585.74,Z 344.9,A -85,B 0,C 180,E1 -564.131,E2 -564.131} C_VEL
LIN {X 0,Y 585.285,Z 341.573,A -85,B 0,C 180,E1 -564.236,E2 -564.236} C_VEL
LIN {X 0,Y 585.629,Z 299.36,A -85,B 0,C 180,E1 -567.4,E2 -567.4} C_VEL
LIN {X 0,Y 585.783,Z 269.109,A -85,B 0,C 180,E1 -569.729,E2 -569.729} C_VEL
LIN {X 0,Y 584.062,Z 263.891,A -85,B 0,C 180,E1 -570.276,E2 -570.276} C_VEL
LIN {X 0,Y 584.09,Z 263.714,A -85,B 0,C 180,E1 -573.45,E2 -573.45} C_VEL
LIN {X 0,Y 584.079,Z 263.731,A -85,B 0,C 180,E1 -576.687,E2 -576.687} C_VEL
LIN {X 0,Y 584.064,Z 263.726,A -85,B 0,C 180,E1 -579.939,E2 -579.939} C_VEL
LIN {X 0,Y 584.093,Z 263.727,A -85,B 0,C 180,E1 -583.08,E2 -583.08} C_VEL
LIN {X 0,Y 584.075,Z 263.728,A -85,B 0,C 180,E1 -586.254,E2 -586.254} C_VEL
LIN {X 0,Y 584.097,Z 263.722,A -85,B 0,C 180,E1 -589.55,E2 -589.55} C_VEL
LIN {X 0,Y 584.086,Z 263.729,A -85,B 0,C 180,E1 -592.822,E2 -592.822} C_VEL
LIN {X 0,Y 584.089,Z 263.727,A -85,B 0,C 180,E1 -596.124,E2 -596.124} C_VEL
LIN {X 0,Y 584.077,Z 263.724,A -85,B 0,C 180,E1 -599.326,E2 -599.326} C_VEL
LIN {X 0,Y 584.073,Z 263.73,A -85,B 0,C 180,E1 -602.691,E2 -602.691} C_VEL
LIN {X 0,Y 584.097,Z 263.725,A -85,B 0,C 180,E1 -605.957,E2 -605.957} C_VEL
LIN {X 0,Y 584.051,Z 263.727,A -85,B 0,C 180,E1 -609.139,E2 -609.139} C_VEL
LIN {X 0,Y 584.074,Z 263.732,A -85,B 0,C 180,E1 -612.361,E2 -612.361} C_VEL
LIN {X 0,Y 584.051,Z 263.726,A -85,B 0,C 180,E1 -615.424,E2 -615.424} C_VEL
LIN {X 0,Y 584.033,Z 263.731,A -85,B 0,C 180,E1 -618.645,E2 -618.645} C_VEL
LIN {X 0,Y 584.067,Z 263.734,A -85,B 0,C 180,E1 -621.683,E2 -621.683} C_VEL
LIN {X 0,Y 584.047,Z 263.964,A -85,B 0,C 180,E1 -622.869,E2 -622.869} C_VEL
LIN {X 0,Y 585.523,Z 269.492,A -85,B 0,C 180,E1 -623.38,E2 -623.38} C_VEL
LIN {X 0,Y 585.652,Z 307.821,A -85,B 0,C 180,E1 -626.279,E2 -626.279} C_VEL
LIN {X 0,Y 585.481,Z 340.59,A -85,B 0,C 180,E1 -628.776,E2 -628.776} C_VEL
LIN {X 0,Y 585.116,Z 381.223,A -85,B 0,C 180,E1 -631.859,E2 -631.859} C_VEL
LIN {X 0,Y 584.848,Z 422.816,A -85,B 0,C 180,E1 -634.952,E2 -634.952} C_VEL
LIN {X 0,Y 584.548,Z 467.504,A -85,B 0,C 180,E1 -638.21,E2 -638.21} C_VEL
LIN {X 0,Y 584.606,Z 472.889,A -85,B 0,C 180,E1 -638.562,E2 -638.562} C_VEL
LIN {X 0,Y 584.78,Z 515.756,A -85,B 0,C 180,E1 -639.109,E2 -639.109} C_VEL
LIN {X 0,Y 584.627,Z 615.439,A -85,B 0,C 180,E1 -640.375,E2 -640.375} C_VEL
LIN {X 0,Y 584.579,Z 632.194,A -85,B 0,C 180,E1 -640.784,E2 -640.784} C_VEL
LIN {X 0,Y 584.479,Z 647.54,A -85,B 0,C 180,E1 -641.344,E2 -641.344} C_VEL
LIN {X 0,Y 584.367,Z 662.663,A -85,B 0,C 180,E1 -642.098,E2 -642.098} C_VEL
LIN {X 0,Y 584.266,Z 676.67,A -85,B 0,C 180,E1 -642.996,E2 -642.996} C_VEL
LIN {X 0,Y 584.154,Z 689.816,A -85,B 0,C 180,E1 -644.065,E2 -644.065} C_VEL
LIN {X 0,Y 584.07,Z 701.828,A -85,B 0,C 180,E1 -645.284,E2 -645.284} C_VEL
LIN {X 0,Y 584.002,Z 712.233,A -85,B 0,C 180,E1 -646.612,E2 -646.612} C_VEL
LIN {X 0,Y 583.96,Z 721.139,A -85,B 0,C 180,E1 -648.052,E2 -648.052} C_VEL
LIN {X 0,Y 583.93,Z 728.436,A -85,B 0,C 180,E1 -649.608,E2 -649.608} C_VEL
LIN {X 0,Y 583.919,Z 733.459,A -85,B 0,C 180,E1 -651.073,E2 -651.073} C_VEL
LIN {X 0,Y 583.914,Z 736.995,A -85,B 0,C 180,E1 -652.659,E2 -652.659} C_VEL
LIN {X 0,Y 583.917,Z 738.77,A -85,B 0,C 180,E1 -654.264,E2 -654.264} C_VEL
LIN {X 0,Y 583.915,Z 738.802,A -85,B 0,C 180,E1 -655.78,E2 -655.78} C_VEL
LIN {X 0,Y 583.915,Z 737.002,A -85,B 0,C 180,E1 -657.425,E2 -657.425} C_VEL
LIN {X 0,Y 583.919,Z 733.555,A -85,B 0,C 180,E1 -658.984,E2 -658.984} C_VEL
LIN {X 0,Y 583.932,Z 728.092,A -85,B 0,C 180,E1 -660.566,E2 -660.566} C_VEL
LIN {X 0,Y 583.959,Z 721.04,A -85,B 0,C 180,E1 -662.057,E2 -662.057} C_VEL
LIN {X 0,Y 584.001,Z 712.401,A -85,B 0,C 180,E1 -663.454,E2 -663.454} C_VEL
LIN {X 0,Y 584.072,Z 701.775,A -85,B 0,C 180,E1 -664.812,E2 -664.812} C_VEL
LIN {X 0,Y 584.153,Z 689.981,A -85,B 0,C 180,E1 -666.01,E2 -666.01} C_VEL
LIN {X 0,Y 584.257,Z 677.416,A -85,B 0,C 180,E1 -667.039,E2 -667.039} C_VEL
LIN {X 0,Y 584.36,Z 663.378,A -85,B 0,C 180,E1 -667.952,E2 -667.952} C_VEL
LIN {X 0,Y 584.47,Z 647.873,A -85,B 0,C 180,E1 -668.731,E2 -668.731} C_VEL
LIN {X 0,Y 584.578,Z 631.879,A -85,B 0,C 180,E1 -669.316,E2 -669.316} C_VEL
LIN {X 0,Y 584.615,Z 614.997,A -85,B 0,C 180,E1 -669.724,E2 -669.724} C_VEL
LIN {X 0,Y 584.627,Z 473.187,A -85,B 0,C 180,E1 -671.521,E2 -671.521} C_VEL
LIN {X 0,Y 584.513,Z 470.309,A -85,B 0,C 180,E1 -671.678,E2 -671.678} C_VEL
LIN {X 0,Y 584.768,Z 429.353,A -85,B 0,C 180,E1 -674.659,E2 -674.659} C_VEL
LIN {X 0,Y 585.047,Z 385.978,A -85,B 0,C 180,E1 -677.875,E2 -677.875} C_VEL
LIN {X 0,Y 585.448,Z 346.351,A -85,B 0,C 180,E1 -680.872,E2 -680.872} C_VEL
LIN {X 0,Y 585.638,Z 312.865,A -85,B 0,C 180,E1 -683.426,E2 -683.426} C_VEL
LIN {X 0,Y 585.451,Z 273.865,A -85,B 0,C 180,E1 -686.344,E2 -686.344} C_VEL
LIN {X 0,Y 585.195,Z 267.775,A -85,B 0,C 180,E1 -686.797,E2 -686.797} C_VEL
LIN {X 0,Y 584.083,Z 263.947,A -85,B 0,C 180,E1 -687.165,E2 -687.165} C_VEL
LIN {X 0,Y 584.101,Z 263.731,A -85,B 0,C 180,E1 -690.236,E2 -690.236} C_VEL
LIN {X 0,Y 584.049,Z 263.729,A -85,B 0,C 180,E1 -693.46,E2 -693.46} C_VEL
LIN {X 0,Y 584.097,Z 263.726,A -85,B 0,C 180,E1 -696.707,E2 -696.707} C_VEL
LIN {X 0,Y 584.061,Z 263.729,A -85,B 0,C 180,E1 -699.873,E2 -699.873} C_VEL
LIN {X 0,Y 584.062,Z 263.726,A -85,B 0,C 180,E1 -703.183,E2 -703.183} C_VEL
LIN {X 0,Y 584.094,Z 263.733,A -85,B 0,C 180,E1 -706.335,E2 -706.335} C_VEL
LIN {X 0,Y 584.052,Z 263.727,A -85,B 0,C 180,E1 -709.544,E2 -709.544} C_VEL
LIN {X 0,Y 584.098,Z 263.726,A -85,B 0,C 180,E1 -712.722,E2 -712.722} C_VEL
LIN {X 0,Y 584.056,Z 263.729,A -85,B 0,C 180,E1 -715.876,E2 -715.876} C_VEL
LIN {X 0,Y 584.086,Z 263.724,A -85,B 0,C 180,E1 -719.117,E2 -719.117} C_VEL
LIN {X 0,Y 584.085,Z 263.731,A -85,B 0,C 180,E1 -722.354,E2 -722.354} C_VEL
LIN {X 0,Y 584.058,Z 263.726,A -85,B 0,C 180,E1 -725.599,E2 -725.599} C_VEL
LIN {X 0,Y 584.097,Z 263.727,A -85,B 0,C 180,E1 -728.763,E2 -728.763} C_VEL
LIN {X 0,Y 584.057,Z 263.728,A -85,B 0,C 180,E1 -731.955,E2 -731.955} C_VEL
LIN {X 0,Y 584.095,Z 263.723,A -85,B 0,C 180,E1 -735.183,E2 -735.183} C_VEL
LIN {X 0,Y 584.089,Z 263.731,A -85,B 0,C 180,E1 -738.501,E2 -738.501} C_VEL
LIN {X 0,Y 584.059,Z 263.726,A -85,B 0,C 180,E1 -741.807,E2 -741.807} C_VEL
LIN {X 0,Y 584.096,Z 263.726,A -85,B 0,C 180,E1 -745.012,E2 -745.012} C_VEL
LIN {X 0,Y 584.062,Z 263.728,A -85,B 0,C 180,E1 -748.195,E2 -748.195} C_VEL
LIN {X 0,Y 584.084,Z 263.723,A -85,B 0,C 180,E1 -751.519,E2 -751.519} C_VEL
LIN {X 0,Y 584.092,Z 263.732,A -85,B 0,C 180,E1 -754.752,E2 -754.752} C_VEL
LIN {X 0,Y 584.063,Z 263.726,A -85,B 0,C 180,E1 -757.921,E2 -757.921} C_VEL
LIN {X 0,Y 584.095,Z 263.728,A -85,B 0,C 180,E1 -761.097,E2 -761.097} C_VEL
LIN {X 0,Y 584.064,Z 263.729,A -85,B 0,C 180,E1 -764.312,E2 -764.312} C_VEL
LIN {X 0,Y 584.092,Z 263.724,A -85,B 0,C 180,E1 -767.59,E2 -767.59} C_VEL
LIN {X 0,Y 584.101,Z 263.731,A -85,B 0,C 180,E1 -770.956,E2 -770.956} C_VEL
LIN {X 0,Y 584.062,Z 263.717,A -85,B 0,C 180,E1 -774.166,E2 -774.166} C_VEL
LIN {X 0,Y 584.093,Z 263.712,A -85,B 0,C 180,E1 -777.374,E2 -777.374} C_VEL
LIN {X 0,Y 584.183,Z 264.259,A -85,B 0,C 180,E1 -777.633,E2 -777.633} C_VEL
LIN {X 0,Y 586.429,Z 270.435,A -85,B 0,C 180,E1 -778.209,E2 -778.209} C_VEL
LIN {X 0,Y 586.03,Z 315.223,A -85,B 0,C 180,E1 -781.176,E2 -781.176} C_VEL
LIN {X 0,Y 586.68,Z 320.862,A -85,B 0,C 180,E1 -781.298,E2 -781.298} C_VEL
LIN {X 0,Y 586.149,Z 549.886,A -85,B 0,C 180,E1 -784.36,E2 -784.36} C_VEL
LIN {X 0,Y 586.038,Z 580.239,A -85,B 0,C 180,E1 -784.804,E2 -784.804} C_VEL
LIN {X 0,Y 585.897,Z 600.76,A -85,B 0,C 180,E1 -785.287,E2 -785.287} C_VEL
LIN {X 0,Y 585.704,Z 621.201,A -85,B 0,C 180,E1 -785.965,E2 -785.965} C_VEL
LIN {X 0,Y 585.478,Z 639.884,A -85,B 0,C 180,E1 -786.767,E2 -786.767} C_VEL
LIN {X 0,Y 585.23,Z 658.759,A -85,B 0,C 180,E1 -787.765,E2 -787.765} C_VEL
LIN {X 0,Y 584.98,Z 677.48,A -85,B 0,C 180,E1 -788.967,E2 -788.967} C_VEL
LIN {X 0,Y 584.755,Z 694.592,A -85,B 0,C 180,E1 -790.279,E2 -790.279} C_VEL
LIN {X 0,Y 584.555,Z 710.114,A -85,B 0,C 180,E1 -791.678,E2 -791.678} C_VEL
LIN {X 0,Y 584.368,Z 725.364,A -85,B 0,C 180,E1 -793.296,E2 -793.296} C_VEL
LIN {X 0,Y 584.207,Z 739.14,A -85,B 0,C 180,E1 -795.024,E2 -795.024} C_VEL
LIN {X 0,Y 584.09,Z 751.3,A -85,B 0,C 180,E1 -796.841,E2 -796.841} C_VEL
LIN {X 0,Y 584.011,Z 761.37,A -85,B 0,C 180,E1 -798.646,E2 -798.646} C_VEL
LIN {X 0,Y 583.957,Z 770.066,A -85,B 0,C 180,E1 -800.54,E2 -800.54} C_VEL
LIN {X 0,Y 583.926,Z 777.192,A -85,B 0,C 180,E1 -802.489,E2 -802.489} C_VEL
LIN {X 0,Y 583.914,Z 782.51,A -85,B 0,C 180,E1 -804.4,E2 -804.4} C_VEL
LIN {X 0,Y 583.907,Z 786.243,A -85,B 0,C 180,E1 -806.369,E2 -806.369} C_VEL
LIN {X 0,Y 583.904,Z 788.374,A -85,B 0,C 180,E1 -808.333,E2 -808.333} C_VEL
LIN {X 0,Y 583.9,Z 788.917,A -85,B 0,C 180,E1 -810.394,E2 -810.394} C_VEL
LIN {X 0,Y 583.905,Z 787.838,A -85,B 0,C 180,E1 -812.356,E2 -812.356} C_VEL
LIN {X 0,Y 583.908,Z 784.971,A -85,B 0,C 180,E1 -814.42,E2 -814.42} C_VEL
LIN {X 0,Y 583.92,Z 780.48,A -85,B 0,C 180,E1 -816.391,E2 -816.391} C_VEL
LIN {X 0,Y 583.943,Z 774.262,A -85,B 0,C 180,E1 -818.37,E2 -818.37} C_VEL
LIN {X 0,Y 583.984,Z 766.173,A -85,B 0,C 180,E1 -820.358,E2 -820.358} C_VEL
LIN {X 0,Y 584.049,Z 756.563,A -85,B 0,C 180,E1 -822.257,E2 -822.257} C_VEL
LIN {X 0,Y 584.148,Z 745.491,A -85,B 0,C 180,E1 -824.068,E2 -824.068} C_VEL
LIN {X 0,Y 584.272,Z 732.93,A -85,B 0,C 180,E1 -825.79,E2 -825.79} C_VEL
LIN {X 0,Y 584.436,Z 718.879,A -85,B 0,C 180,E1 -827.422,E2 -827.422} C_VEL
LIN {X 0,Y 584.624,Z 703.836,A -85,B 0,C 180,E1 -828.912,E2 -828.912} C_VEL
LIN {X 0,Y 584.844,Z 687.279,A -85,B 0,C 180,E1 -830.308,E2 -830.308} C_VEL
LIN {X 0,Y 585.085,Z 669.738,A -85,B 0,C 180,E1 -831.557,E2 -831.557} C_VEL
LIN {X 0,Y 585.339,Z 651.251,A -85,B 0,C 180,E1 -832.657,E2 -832.657} C_VEL
LIN {X 0,Y 585.578,Z 633.055,A -85,B 0,C 180,E1 -833.551,E2 -833.551} C_VEL
LIN {X 0,Y 585.764,Z 613.629,A -85,B 0,C 180,E1 -834.308,E2 -834.308} C_VEL
LIN {X 0,Y 585.938,Z 593.746,A -85,B 0,C 180,E1 -834.896,E2 -834.896} C_VEL
LIN {X 0,Y 586.085,Z 572.695,A -85,B 0,C 180,E1 -835.325,E2 -835.325} C_VEL
LIN {X 0,Y 586.658,Z 330.991,A -85,B 0,C 180,E1 -838.565,E2 -838.565} C_VEL
LIN {X 0,Y 586.455,Z 317.862,A -85,B 0,C 180,E1 -838.755,E2 -838.755} C_VEL
LIN {X 0,Y 586.013,Z 314.36,A -85,B 0,C 180,E1 -838.873,E2 -838.873} C_VEL
LIN {X 0,Y 586.423,Z 270.398,A -85,B 0,C 180,E1 -841.794,E2 -841.794} C_VEL
LIN {X 0,Y 584.143,Z 264.042,A -85,B 0,C 180,E1 -842.396,E2 -842.396} C_VEL
LIN {X 0,Y 584.087,Z 263.723,A -85,B 0,C 180,E1 -843.167,E2 -843.167} C_VEL
LIN {X 0,Y 584.097,Z 263.726,A -85,B 0,C 180,E1 -846.442,E2 -846.442} C_VEL
LIN {X 0,Y 584.058,Z 263.729,A -85,B 0,C 180,E1 -849.684,E2 -849.684} C_VEL
LIN {X 0,Y 584.097,Z 263.731,A -85,B 0,C 180,E1 -852.891,E2 -852.891} C_VEL
LIN {X 0,Y 584.057,Z 263.728,A -85,B 0,C 180,E1 -855.973,E2 -855.973} C_VEL
LIN {X 0,Y 584.074,Z 263.732,A -85,B 0,C 180,E1 -859.291,E2 -859.291} C_VEL
LIN {X 0,Y 584.086,Z 263.726,A -85,B 0,C 180,E1 -862.453,E2 -862.453} C_VEL
LIN {X 0,Y 584.051,Z 263.732,A -85,B 0,C 180,E1 -865.605,E2 -865.605} C_VEL
LIN {X 0,Y 584.099,Z 263.724,A -85,B 0,C 180,E1 -868.757,E2 -868.757} C_VEL
LIN {X 0,Y 584.072,Z 263.937,A -85,B 0,C 180,E1 -869.826,E2 -869.826} C_VEL
LIN {X 0,Y 585.933,Z 270.168,A -85,B 0,C 180,E1 -870.452,E2 -870.452} C_VEL
LIN {X 0,Y 585.51,Z 310.492,A -85,B 0,C 180,E1 -873.532,E2 -873.532} C_VEL
LIN {X 0,Y 585.352,Z 342.589,A -85,B 0,C 180,E1 -875.906,E2 -875.906} C_VEL
LIN {X 0,Y 585.885,Z 347.766,A -85,B 0,C 180,E1 -876.003,E2 -876.003} C_VEL
LIN {X 0,Y 585.445,Z 559.888,A -85,B 0,C 180,E1 -878.773,E2 -878.773} C_VEL
LIN {X 0,Y 585.327,Z 579.62,A -85,B 0,C 180,E1 -879.224,E2 -879.224} C_VEL
LIN {X 0,Y 585.167,Z 598.8,A -85,B 0,C 180,E1 -879.861,E2 -879.861} C_VEL
LIN {X 0,Y 584.985,Z 617.38,A -85,B 0,C 180,E1 -880.682,E2 -880.682} C_VEL
LIN {X 0,Y 584.796,Z 634.971,A -85,B 0,C 180,E1 -881.664,E2 -881.664} C_VEL
LIN {X 0,Y 584.604,Z 651.393,A -85,B 0,C 180,E1 -882.79,E2 -882.79} C_VEL
LIN {X 0,Y 584.428,Z 666.638,A -85,B 0,C 180,E1 -884.048,E2 -884.048} C_VEL
LIN {X 0,Y 584.27,Z 680.625,A -85,B 0,C 180,E1 -885.43,E2 -885.43} C_VEL
LIN {X 0,Y 584.146,Z 693.461,A -85,B 0,C 180,E1 -886.942,E2 -886.942} C_VEL
LIN {X 0,Y 584.056,Z 704.794,A -85,B 0,C 180,E1 -888.546,E2 -888.546} C_VEL
LIN {X 0,Y 583.982,Z 714.637,A -85,B 0,C 180,E1 -890.241,E2 -890.241} C_VEL
LIN {X 0,Y 583.946,Z 722.963,A -85,B 0,C 180,E1 -892.028,E2 -892.028} C_VEL
LIN {X 0,Y 583.919,Z 729.705,A -85,B 0,C 180,E1 -893.906,E2 -893.906} C_VEL
LIN {X 0,Y 583.909,Z 734.533,A -85,B 0,C 180,E1 -895.778,E2 -895.778} C_VEL
LIN {X 0,Y 583.914,Z 737.566,A -85,B 0,C 180,E1 -897.645,E2 -897.645} C_VEL
LIN {X 0,Y 583.905,Z 738.907,A -85,B 0,C 180,E1 -899.608,E2 -899.608} C_VEL
LIN {X 0,Y 583.912,Z 738.464,A -85,B 0,C 180,E1 -901.472,E2 -901.472} C_VEL
LIN {X 0,Y 583.915,Z 736.322,A -85,B 0,C 180,E1 -903.344,E2 -903.344} C_VEL
LIN {X 0,Y 583.92,Z 732.452,A -85,B 0,C 180,E1 -905.207,E2 -905.207} C_VEL
LIN {X 0,Y 583.936,Z 726.727,A -85,B 0,C 180,E1 -907.082,E2 -907.082} C_VEL
LIN {X 0,Y 583.966,Z 719.004,A -85,B 0,C 180,E1 -908.964,E2 -908.964} C_VEL
LIN {X 0,Y 584.018,Z 709.624,A -85,B 0,C 180,E1 -910.756,E2 -910.756} C_VEL
LIN {X 0,Y 584.095,Z 699.324,A -85,B 0,C 180,E1 -912.356,E2 -912.356} C_VEL
LIN {X 0,Y 584.108,Z 698.186,A -85,B 0,C 180,E1 -912.518,E2 -912.518} C_VEL
LIN {X 0,Y 583.191,Z 693.811,A -85,B 0,C 180,E1 -913.141,E2 -913.141} C_VEL
LIN {X 0,Y 577.405,Z 682.292,A -85,B 0,C 180,E1 -914.671,E2 -914.671} C_VEL
LIN {X 0,Y 576.462,Z 677.121,A -85,B 0,C 180,E1 -915.24,E2 -915.24} C_VEL
LIN {X 0,Y 576.677,Z 662.603,A -85,B 0,C 180,E1 -916.624,E2 -916.624} C_VEL
LIN {X 0,Y 576.922,Z 647.026,A -85,B 0,C 180,E1 -917.864,E2 -917.864} C_VEL
LIN {X 0,Y 577.169,Z 630.739,A -85,B 0,C 180,E1 -918.938,E2 -918.938} C_VEL
LIN {X 0,Y 577.424,Z 613.289,A -85,B 0,C 180,E1 -919.874,E2 -919.874} C_VEL
LIN {X 0,Y 577.656,Z 595.368,A -85,B 0,C 180,E1 -920.634,E2 -920.634} C_VEL
LIN {X 0,Y 577.86,Z 576.166,A -85,B 0,C 180,E1 -921.242,E2 -921.242} C_VEL
LIN {X 0,Y 578.008,Z 557.027,A -85,B 0,C 180,E1 -921.652,E2 -921.652} C_VEL
LIN {X 0,Y 578.445,Z 346.121,A -85,B 0,C 180,E1 -924.438,E2 -924.438} C_VEL
LIN {X 0,Y 577.781,Z 342.045,A -85,B 0,C 180,E1 -924.54,E2 -924.54} C_VEL
LIN {X 0,Y 578.245,Z 300.128,A -85,B 0,C 180,E1 -927.719,E2 -927.719} C_VEL
LIN {X 0,Y 578.472,Z 272.066,A -85,B 0,C 180,E1 -929.908,E2 -929.908} C_VEL
LIN {X 0,Y 576.148,Z 264.916,A -85,B 0,C 180,E1 -930.647,E2 -930.647} C_VEL
LIN {X 0,Y 576.111,Z 264.701,A -85,B 0,C 180,E1 -933.976,E2 -933.976} C_VEL
LIN {X 0,Y 576.16,Z 264.716,A -85,B 0,C 180,E1 -937.151,E2 -937.151} C_VEL
LIN {X 0,Y 576.128,Z 264.718,A -85,B 0,C 180,E1 -940.369,E2 -940.369} C_VEL
LIN {X 0,Y 576.145,Z 264.713,A -85,B 0,C 180,E1 -943.686,E2 -943.686} C_VEL
LIN {X 0,Y 576.15,Z 264.717,A -85,B 0,C 180,E1 -946.998,E2 -946.998} C_VEL
LIN {X 0,Y 576.144,Z 264.717,A -85,B 0,C 180,E1 -950.247,E2 -950.247} C_VEL
LIN {X 0,Y 576.158,Z 264.711,A -85,B 0,C 180,E1 -953.593,E2 -953.593} C_VEL
LIN {X 0,Y 576.138,Z 264.717,A -85,B 0,C 180,E1 -956.861,E2 -956.861} C_VEL
LIN {X 0,Y 576.155,Z 264.716,A -85,B 0,C 180,E1 -960.127,E2 -960.127} C_VEL
LIN {X 0,Y 576.134,Z 264.714,A -85,B 0,C 180,E1 -963.4,E2 -963.4} C_VEL
LIN {X 0,Y 576.125,Z 264.719,A -85,B 0,C 180,E1 -966.69,E2 -966.69} C_VEL
LIN {X 0,Y 576.161,Z 264.715,A -85,B 0,C 180,E1 -969.902,E2 -969.902} C_VEL
LIN {X 0,Y 576.102,Z 264.719,A -85,B 0,C 180,E1 -973.047,E2 -973.047} C_VEL
LIN {X 0,Y 576.136,Z 264.713,A -85,B 0,C 180,E1 -976.245,E2 -976.245} C_VEL
LIN {X 0,Y 576.096,Z 264.719,A -85,B 0,C 180,E1 -979.297,E2 -979.297} C_VEL
LIN {X 0,Y 576.102,Z 264.798,A -85,B 0,C 180,E1 -982.52,E2 -982.52} C_VEL
LIN {X 0,Y 576.549,Z 266.601,A -85,B 0,C 180,E1 -982.738,E2 -982.738} C_VEL
LIN {X 0,Y 578.054,Z 272.367,A -85,B 0,C 180,E1 -983.244,E2 -983.244} C_VEL
LIN {X 0,Y 578.093,Z 311.497,A -85,B 0,C 180,E1 -986.231,E2 -986.231} C_VEL
LIN {X 0,Y 577.913,Z 352.736,A -85,B 0,C 180,E1 -989.355,E2 -989.355} C_VEL
LIN {X 0,Y 577.434,Z 393.635,A -85,B 0,C 180,E1 -992.48,E2 -992.48} C_VEL
LIN {X 0,Y 577.022,Z 438.206,A -85,B 0,C 180,E1 -995.817,E2 -995.817} C_VEL
LIN {X 0,Y 576.787,Z 472.434,A -85,B 0,C 180,E1 -998.321,E2 -998.321} C_VEL
LIN {X 0,Y 577.159,Z 479.84,A -85,B 0,C 180,E1 -998.436,E2 -998.436} C_VEL
LIN {X 0,Y 576.884,Z 615.467,A -85,B 0,C 180,E1 -1000.174,E2 -1000.174} C_VEL
LIN {X 0,Y 576.81,Z 632.149,A -85,B 0,C 180,E1 -1000.587,E2 -1000.587} C_VEL
LIN {X 0,Y 576.685,Z 647.298,A -85,B 0,C 180,E1 -1001.145,E2 -1001.145} C_VEL
LIN {X 0,Y 576.528,Z 662.503,A -85,B 0,C 180,E1 -1001.909,E2 -1001.909} C_VEL
LIN {X 0,Y 576.388,Z 676.649,A -85,B 0,C 180,E1 -1002.828,E2 -1002.828} C_VEL
LIN {X 0,Y 576.244,Z 689.721,A -85,B 0,C 180,E1 -1003.904,E2 -1003.904} C_VEL
LIN {X 0,Y 576.131,Z 701.3,A -85,B 0,C 180,E1 -1005.088,E2 -1005.088} C_VEL
LIN {X 0,Y 576.037,Z 711.807,A -85,B 0,C 180,E1 -1006.434,E2 -1006.434} C_VEL
LIN {X 0,Y 575.977,Z 720.813,A -85,B 0,C 180,E1 -1007.893,E2 -1007.893} C_VEL
LIN {X 0,Y 575.939,Z 727.754,A -85,B 0,C 180,E1 -1009.364,E2 -1009.364} C_VEL
LIN {X 0,Y 575.923,Z 733.265,A -85,B 0,C 180,E1 -1010.954,E2 -1010.954} C_VEL
LIN {X 0,Y 575.917,Z 736.857,A -85,B 0,C 180,E1 -1012.538,E2 -1012.538} C_VEL
LIN {X 0,Y 575.918,Z 738.726,A -85,B 0,C 180,E1 -1014.186,E2 -1014.186} C_VEL
LIN {X 0,Y 575.915,Z 738.844,A -85,B 0,C 180,E1 -1015.722,E2 -1015.722} C_VEL
LIN {X 0,Y 575.915,Z 737.109,A -85,B 0,C 180,E1 -1017.39,E2 -1017.39} C_VEL
LIN {X 0,Y 575.92,Z 733.738,A -85,B 0,C 180,E1 -1018.97,E2 -1018.97} C_VEL
LIN {X 0,Y 575.938,Z 728.373,A -85,B 0,C 180,E1 -1020.573,E2 -1020.573} C_VEL
LIN {X 0,Y 575.973,Z 721.338,A -85,B 0,C 180,E1 -1022.097,E2 -1022.097} C_VEL
LIN {X 0,Y 576.029,Z 712.879,A -85,B 0,C 180,E1 -1023.501,E2 -1023.501} C_VEL
LIN {X 0,Y 576.121,Z 702.422,A -85,B 0,C 180,E1 -1024.871,E2 -1024.871} C_VEL
LIN {X 0,Y 576.233,Z 690.822,A -85,B 0,C 180,E1 -1026.084,E2 -1026.084} C_VEL
LIN {X 0,Y 576.376,Z 677.75,A -85,B 0,C 180,E1 -1027.18,E2 -1027.18} C_VEL
LIN {X 0,Y 576.508,Z 664.634,A -85,B 0,C 180,E1 -1028.057,E2 -1028.057} C_VEL
LIN {X 0,Y 576.648,Z 649.686,A -85,B 0,C 180,E1 -1028.838,E2 -1028.838} C_VEL
LIN {X 0,Y 576.795,Z 633.926,A -85,B 0,C 180,E1 -1029.447,E2 -1029.447} C_VEL
LIN {X 0,Y 576.868,Z 617.413,A -85,B 0,C 180,E1 -1029.878,E2 -1029.878} C_VEL
LIN {X 0,Y 576.913,Z 591.139,A -85,B 0,C 180,E1 -1030.25,E2 -1030.25} C_VEL
LIN {X 0,Y 576.946,Z 473.984,A -85,B 0,C 180,E1 -1031.735,E2 -1031.735} C_VEL
LIN {X 0,Y 576.748,Z 471.856,A -85,B 0,C 180,E1 -1031.801,E2 -1031.801} C_VEL
LIN {X 0,Y 577.064,Z 431.503,A -85,B 0,C 180,E1 -1034.771,E2 -1034.771} C_VEL
LIN {X 0,Y 577.457,Z 388.314,A -85,B 0,C 180,E1 -1038.014,E2 -1038.014} C_VEL
LIN {X 0,Y 577.962,Z 348.869,A -85,B 0,C 180,E1 -1041.034,E2 -1041.034} C_VEL
LIN {X 0,Y 578.032,Z 306.453,A -85,B 0,C 180,E1 -1044.22,E2 -1044.22} C_VEL
LIN {X 0,Y 577.91,Z 276.15,A -85,B 0,C 180,E1 -1046.501,E2 -1046.501} C_VEL
LIN {X 0,Y 577.638,Z 270.109,A -85,B 0,C 180,E1 -1046.958,E2 -1046.958} C_VEL
LIN {X 0,Y 576.147,Z 264.988,A -85,B 0,C 180,E1 -1047.438,E2 -1047.438} C_VEL
LIN {X 0,Y 576.136,Z 264.722,A -85,B 0,C 180,E1 -1050.012,E2 -1050.012} C_VEL
LIN {X 0,Y 576.113,Z 264.717,A -85,B 0,C 180,E1 -1053.288,E2 -1053.288} C_VEL
LIN {X 0,Y 576.161,Z 264.718,A -85,B 0,C 180,E1 -1056.475,E2 -1056.475} C_VEL
LIN {X 0,Y 576.113,Z 264.717,A -85,B 0,C 180,E1 -1059.689,E2 -1059.689} C_VEL
LIN {X 0,Y 576.14,Z 264.715,A -85,B 0,C 180,E1 -1062.979,E2 -1062.979} C_VEL
LIN {X 0,Y 576.139,Z 264.72,A -85,B 0,C 180,E1 -1066.143,E2 -1066.143} C_VEL
LIN {X 0,Y 576.117,Z 264.715,A -85,B 0,C 180,E1 -1069.399,E2 -1069.399} C_VEL
LIN {X 0,Y 576.16,Z 264.717,A -85,B 0,C 180,E1 -1072.621,E2 -1072.621} C_VEL
LIN {X 0,Y 576.116,Z 264.717,A -85,B 0,C 180,E1 -1075.82,E2 -1075.82} C_VEL
LIN {X 0,Y 576.148,Z 264.713,A -85,B 0,C 180,E1 -1079.105,E2 -1079.105} C_VEL
LIN {X 0,Y 576.149,Z 264.72,A -85,B 0,C 180,E1 -1082.387,E2 -1082.387} C_VEL
LIN {X 0,Y 576.117,Z 264.716,A -85,B 0,C 180,E1 -1085.677,E2 -1085.677} C_VEL
LIN {X 0,Y 576.159,Z 264.714,A -85,B 0,C 180,E1 -1088.885,E2 -1088.885} C_VEL
LIN {X 0,Y 576.124,Z 264.718,A -85,B 0,C 180,E1 -1092.122,E2 -1092.122} C_VEL
LIN {X 0,Y 576.131,Z 264.713,A -85,B 0,C 180,E1 -1095.501,E2 -1095.501} C_VEL
LIN {X 0,Y 576.159,Z 264.719,A -85,B 0,C 180,E1 -1098.726,E2 -1098.726} C_VEL
LIN {X 0,Y 576.119,Z 264.715,A -85,B 0,C 180,E1 -1101.909,E2 -1101.909} C_VEL
LIN {X 0,Y 576.158,Z 264.713,A -85,B 0,C 180,E1 -1105.161,E2 -1105.161} C_VEL
LIN {X 0,Y 576.133,Z 264.718,A -85,B 0,C 180,E1 -1108.393,E2 -1108.393} C_VEL
LIN {X 0,Y 576.129,Z 264.714,A -85,B 0,C 180,E1 -1111.75,E2 -1111.75} C_VEL
LIN {X 0,Y 576.157,Z 264.717,A -85,B 0,C 180,E1 -1115.008,E2 -1115.008} C_VEL
LIN {X 0,Y 576.122,Z 264.716,A -85,B 0,C 180,E1 -1118.173,E2 -1118.173} C_VEL
LIN {X 0,Y 576.159,Z 264.712,A -85,B 0,C 180,E1 -1121.439,E2 -1121.439} C_VEL
LIN {X 0,Y 576.155,Z 264.72,A -85,B 0,C 180,E1 -1124.795,E2 -1124.795} C_VEL
LIN {X 0,Y 576.125,Z 264.717,A -85,B 0,C 180,E1 -1128.118,E2 -1128.118} C_VEL
LIN {X 0,Y 576.156,Z 264.716,A -85,B 0,C 180,E1 -1131.345,E2 -1131.345} C_VEL
LIN {X 0,Y 576.131,Z 264.701,A -85,B 0,C 180,E1 -1134.576,E2 -1134.576} C_VEL
LIN {X 0,Y 576.191,Z 264.963,A -85,B 0,C 180,E1 -1137.153,E2 -1137.153} C_VEL
LIN {X 0,Y 579.319,Z 273.816,A -85,B 0,C 180,E1 -1138.006,E2 -1138.006} C_VEL
LIN {X 0,Y 578.843,Z 315.684,A -85,B 0,C 180,E1 -1140.796,E2 -1140.796} C_VEL
LIN {X 0,Y 579.658,Z 322.135,A -85,B 0,C 180,E1 -1140.935,E2 -1140.935} C_VEL
LIN {X 0,Y 578.931,Z 551.159,A -85,B 0,C 180,E1 -1144.034,E2 -1144.034} C_VEL
LIN {X 0,Y 578.782,Z 580.563,A -85,B 0,C 180,E1 -1144.473,E2 -1144.473} C_VEL
LIN {X 0,Y 578.596,Z 600.975,A -85,B 0,C 180,E1 -1144.96,E2 -1144.96} C_VEL
LIN {X 0,Y 578.344,Z 620.736,A -85,B 0,C 180,E1 -1145.622,E2 -1145.622} C_VEL
LIN {X 0,Y 578.032,Z 640.069,A -85,B 0,C 180,E1 -1146.459,E2 -1146.459} C_VEL
LIN {X 0,Y 577.706,Z 658.883,A -85,B 0,C 180,E1 -1147.467,E2 -1147.467} C_VEL
LIN {X 0,Y 577.367,Z 677.791,A -85,B 0,C 180,E1 -1148.698,E2 -1148.698} C_VEL
LIN {X 0,Y 577.055,Z 695.027,A -85,B 0,C 180,E1 -1150.043,E2 -1150.043} C_VEL
LIN {X 0,Y 576.768,Z 710.925,A -85,B 0,C 180,E1 -1151.505,E2 -1151.505} C_VEL
LIN {X 0,Y 576.53,Z 725.365,A -85,B 0,C 180,E1 -1153.062,E2 -1153.062} C_VEL
LIN {X 0,Y 576.317,Z 739.139,A -85,B 0,C 180,E1 -1154.814,E2 -1154.814} C_VEL
LIN {X 0,Y 576.152,Z 751.299,A -85,B 0,C 180,E1 -1156.657,E2 -1156.657} C_VEL
LIN {X 0,Y 576.044,Z 761.371,A -85,B 0,C 180,E1 -1158.487,E2 -1158.487} C_VEL
LIN {X 0,Y 575.975,Z 770.066,A -85,B 0,C 180,E1 -1160.408,E2 -1160.408} C_VEL
LIN {X 0,Y 575.943,Z 776.994,A -85,B 0,C 180,E1 -1162.319,E2 -1162.319} C_VEL
LIN {X 0,Y 575.92,Z 782.511,A -85,B 0,C 180,E1 -1164.322,E2 -1164.322} C_VEL
LIN {X 0,Y 575.91,Z 786.243,A -85,B 0,C 180,E1 -1166.318,E2 -1166.318} C_VEL
LIN {X 0,Y 575.905,Z 788.374,A -85,B 0,C 180,E1 -1168.31,E2 -1168.31} C_VEL
LIN {X 0,Y 575.9,Z 788.917,A -85,B 0,C 180,E1 -1170.399,E2 -1170.399} C_VEL
LIN {X 0,Y 575.905,Z 787.838,A -85,B 0,C 180,E1 -1172.389,E2 -1172.389} C_VEL
LIN {X 0,Y 575.911,Z 784.971,A -85,B 0,C 180,E1 -1174.482,E2 -1174.482} C_VEL
LIN {X 0,Y 575.924,Z 780.481,A -85,B 0,C 180,E1 -1176.48,E2 -1176.48} C_VEL
LIN {X 0,Y 575.954,Z 774.262,A -85,B 0,C 180,E1 -1178.487,E2 -1178.487} C_VEL
LIN {X 0,Y 576.006,Z 766.174,A -85,B 0,C 180,E1 -1180.503,E2 -1180.503} C_VEL
LIN {X 0,Y 576.095,Z 756.562,A -85,B 0,C 180,E1 -1182.429,E2 -1182.429} C_VEL
LIN {X 0,Y 576.234,Z 745.489,A -85,B 0,C 180,E1 -1184.265,E2 -1184.265} C_VEL
LIN {X 0,Y 576.418,Z 732.554,A -85,B 0,C 180,E1 -1186.061,E2 -1186.061} C_VEL
LIN {X 0,Y 576.65,Z 717.952,A -85,B 0,C 180,E1 -1187.769,E2 -1187.769} C_VEL
LIN {X 0,Y 576.931,Z 702.17,A -85,B 0,C 180,E1 -1189.331,E2 -1189.331} C_VEL
LIN {X 0,Y 577.235,Z 685.35,A -85,B 0,C 180,E1 -1190.741,E2 -1190.741} C_VEL
LIN {X 0,Y 577.543,Z 668.135,A -85,B 0,C 180,E1 -1191.96,E2 -1191.96} C_VEL
LIN {X 0,Y 577.869,Z 649.262,A -85,B 0,C 180,E1 -1193.074,E2 -1193.074} C_VEL
LIN {X 0,Y 578.193,Z 629.24,A -85,B 0,C 180,E1 -1194.033,E2 -1194.033} C_VEL
LIN {X 0,Y 578.494,Z 609.339,A -85,B 0,C 180,E1 -1194.781,E2 -1194.781} C_VEL
LIN {X 0,Y 578.736,Z 589.022,A -85,B 0,C 180,E1 -1195.35,E2 -1195.35} C_VEL
LIN {X 0,Y 578.868,Z 568.031,A -85,B 0,C 180,E1 -1195.738,E2 -1195.738} C_VEL
LIN {X 0,Y 579.622,Z 333.536,A -85,B 0,C 180,E1 -1198.909,E2 -1198.909} C_VEL
LIN {X 0,Y 579.439,Z 319.158,A -85,B 0,C 180,E1 -1199.119,E2 -1199.119} C_VEL
LIN {X 0,Y 578.776,Z 314.495,A -85,B 0,C 180,E1 -1199.261,E2 -1199.261} C_VEL
LIN {X 0,Y 579.284,Z 273.474,A -85,B 0,C 180,E1 -1202.02,E2 -1202.02} C_VEL
LIN {X 0,Y 576.188,Z 264.941,A -85,B 0,C 180,E1 -1202.848,E2 -1202.848} C_VEL
LIN {X 0,Y 576.132,Z 264.717,A -85,B 0,C 180,E1 -1206.039,E2 -1206.039} C_VEL
LIN {X 0,Y 576.128,Z 264.72,A -85,B 0,C 180,E1 -1209.44,E2 -1209.44} C_VEL
LIN {X 0,Y 576.16,Z 264.716,A -85,B 0,C 180,E1 -1212.625,E2 -1212.625} C_VEL
LIN {X 0,Y 576.115,Z 264.718,A -85,B 0,C 180,E1 -1215.789,E2 -1215.789} C_VEL
LIN {X 0,Y 576.161,Z 264.72,A -85,B 0,C 180,E1 -1219.017,E2 -1219.017} C_VEL
LIN {X 0,Y 576.126,Z 264.717,A -85,B 0,C 180,E1 -1222.221,E2 -1222.221} C_VEL
LIN {X 0,Y 576.115,Z 264.722,A -85,B 0,C 180,E1 -1225.544,E2 -1225.544} C_VEL
LIN {X 0,Y 576.16,Z 264.709,A -85,B 0,C 180,E1 -1228.743,E2 -1228.743} C_VEL
LIN {X 0,Y 576.164,Z 265.039,A -85,B 0,C 180,E1 -1229.468,E2 -1229.468} C_VEL
LIN {X 0,Y 578.615,Z 273.057,A -85,B 0,C 180,E1 -1230.268,E2 -1230.268} C_VEL
LIN {X 0,Y 578.061,Z 313.726,A -85,B 0,C 180,E1 -1233.412,E2 -1233.412} C_VEL
LIN {X 0,Y 577.847,Z 342.642,A -85,B 0,C 180,E1 -1235.573,E2 -1235.573} C_VEL
LIN {X 0,Y 578.574,Z 348.669,A -85,B 0,C 180,E1 -1235.691,E2 -1235.691} C_VEL
LIN {X 0,Y 577.985,Z 559.915,A -85,B 0,C 180,E1 -1238.486,E2 -1238.486} C_VEL
LIN {X 0,Y 577.826,Z 579.635,A -85,B 0,C 180,E1 -1238.942,E2 -1238.942} C_VEL
LIN {X 0,Y 577.628,Z 598.179,A -85,B 0,C 180,E1 -1239.56,E2 -1239.56} C_VEL
LIN {X 0,Y 577.387,Z 616.468,A -85,B 0,C 180,E1 -1240.37,E2 -1240.37} C_VEL
LIN {X 0,Y 577.127,Z 634.544,A -85,B 0,C 180,E1 -1241.383,E2 -1241.383} C_VEL
LIN {X 0,Y 576.872,Z 650.743,A -85,B 0,C 180,E1 -1242.5,E2 -1242.5} C_VEL
LIN {X 0,Y 576.626,Z 666.249,A -85,B 0,C 180,E1 -1243.79,E2 -1243.79} C_VEL
LIN {X 0,Y 576.407,Z 680.631,A -85,B 0,C 180,E1 -1245.227,E2 -1245.227} C_VEL
LIN {X 0,Y 576.239,Z 693.478,A -85,B 0,C 180,E1 -1246.761,E2 -1246.761} C_VEL
LIN {X 0,Y 576.105,Z 704.801,A -85,B 0,C 180,E1 -1248.386,E2 -1248.386} C_VEL
LIN {X 0,Y 576.012,Z 714.642,A -85,B 0,C 180,E1 -1250.105,E2 -1250.105} C_VEL
LIN {X 0,Y 575.955,Z 722.965,A -85,B 0,C 180,E1 -1251.917,E2 -1251.917} C_VEL
LIN {X 0,Y 575.926,Z 729.708,A -85,B 0,C 180,E1 -1253.821,E2 -1253.821} C_VEL
LIN {X 0,Y 575.91,Z 734.537,A -85,B 0,C 180,E1 -1255.719,E2 -1255.719} C_VEL
LIN {X 0,Y 575.914,Z 737.569,A -85,B 0,C 180,E1 -1257.612,E2 -1257.612} C_VEL
LIN {X 0,Y 575.908,Z 738.885,A -85,B 0,C 180,E1 -1259.503,E2 -1259.503} C_VEL
LIN {X 0,Y 575.912,Z 738.465,A -85,B 0,C 180,E1 -1261.493,E2 -1261.493} C_VEL
LIN {X 0,Y 575.913,Z 736.334,A -85,B 0,C 180,E1 -1263.384,E2 -1263.384} C_VEL
LIN {X 0,Y 575.92,Z 732.453,A -85,B 0,C 180,E1 -1265.28,E2 -1265.28} C_VEL
LIN {X 0,Y 575.944,Z 726.725,A -85,B 0,C 180,E1 -1267.181,E2 -1267.181} C_VEL
LIN {X 0,Y 575.985,Z 719.001,A -85,B 0,C 180,E1 -1269.089,E2 -1269.089} C_VEL
LIN {X 0,Y 576.061,Z 709.623,A -85,B 0,C 180,E1 -1270.906,E2 -1270.906} C_VEL
LIN {X 0,Y 576.172,Z 698.969,A -85,B 0,C 180,E1 -1272.58,E2 -1272.58} C_VEL
LIN {X 0,Y 576.325,Z 686.817,A -85,B 0,C 180,E1 -1274.16,E2 -1274.16} C_VEL
LIN {X 0,Y 576.462,Z 677.121,A -85,B 0,C 180,E1 -1275.24,E2 -1275.24} C_VEL
LIN {X 0,Y 575.534,Z 671.912,A -85,B 0,C 180,E1 -1275.797,E2 -1275.797} C_VEL
LIN {X 0,Y 569.928,Z 658.431,A -85,B 0,C 180,E1 -1277.19,E2 -1277.19} C_VEL
LIN {X 0,Y 569.093,Z 652.545,A -85,B 0,C 180,E1 -1277.695,E2 -1277.695} C_VEL
LIN {X 0,Y 569.414,Z 636.354,A -85,B 0,C 180,E1 -1278.851,E2 -1278.851} C_VEL
LIN {X 0,Y 569.729,Z 619.186,A -85,B 0,C 180,E1 -1279.852,E2 -1279.852} C_VEL
LIN {X 0,Y 570.031,Z 600.967,A -85,B 0,C 180,E1 -1280.698,E2 -1280.698} C_VEL
LIN {X 0,Y 570.301,Z 582.037,A -85,B 0,C 180,E1 -1281.367,E2 -1281.367} C_VEL
LIN {X 0,Y 570.505,Z 562.731,A -85,B 0,C 180,E1 -1281.845,E2 -1281.845} C_VEL
LIN {X 0,Y 570.667,Z 532.892,A -85,B 0,C 180,E1 -1282.282,E2 -1282.282} C_VEL
LIN {X 0,Y 571.13,Z 347.18,A -85,B 0,C 180,E1 -1284.757,E2 -1284.757} C_VEL
LIN {X 0,Y 570.292,Z 342.045,A -85,B 0,C 180,E1 -1284.884,E2 -1284.884} C_VEL
LIN {X 0,Y 570.913,Z 299.398,A -85,B 0,C 180,E1 -1288.164,E2 -1288.164} C_VEL
LIN {X 0,Y 571.231,Z 275.144,A -85,B 0,C 180,E1 -1290.078,E2 -1290.078} C_VEL
LIN {X 0,Y 568.25,Z 265.922,A -85,B 0,C 180,E1 -1291.034,E2 -1291.034} C_VEL
LIN {X 0,Y 568.171,Z 265.688,A -85,B 0,C 180,E1 -1294.273,E2 -1294.273} C_VEL
LIN {X 0,Y 568.213,Z 265.703,A -85,B 0,C 180,E1 -1297.506,E2 -1297.506} C_VEL
LIN {X 0,Y 568.222,Z 265.708,A -85,B 0,C 180,E1 -1300.83,E2 -1300.83} C_VEL
LIN {X 0,Y 568.192,Z 265.705,A -85,B 0,C 180,E1 -1304.112,E2 -1304.112} C_VEL
LIN {X 0,Y 568.216,Z 265.702,A -85,B 0,C 180,E1 -1307.353,E2 -1307.353} C_VEL
LIN {X 0,Y 568.216,Z 265.708,A -85,B 0,C 180,E1 -1310.737,E2 -1310.737} C_VEL
LIN {X 0,Y 568.207,Z 265.704,A -85,B 0,C 180,E1 -1314.043,E2 -1314.043} C_VEL
LIN {X 0,Y 568.201,Z 265.702,A -85,B 0,C 180,E1 -1317.3,E2 -1317.3} C_VEL
LIN {X 0,Y 568.198,Z 265.706,A -85,B 0,C 180,E1 -1320.711,E2 -1320.711} C_VEL
LIN {X 0,Y 568.219,Z 265.705,A -85,B 0,C 180,E1 -1324.013,E2 -1324.013} C_VEL
LIN {X 0,Y 568.181,Z 265.705,A -85,B 0,C 180,E1 -1327.238,E2 -1327.238} C_VEL
LIN {X 0,Y 568.182,Z 265.708,A -85,B 0,C 180,E1 -1330.602,E2 -1330.602} C_VEL
LIN {X 0,Y 568.211,Z 265.706,A -85,B 0,C 180,E1 -1333.752,E2 -1333.752} C_VEL
LIN {X 0,Y 568.153,Z 265.708,A -85,B 0,C 180,E1 -1336.877,E2 -1336.877} C_VEL
LIN {X 0,Y 568.205,Z 265.697,A -85,B 0,C 180,E1 -1340.069,E2 -1340.069} C_VEL
LIN {X 0,Y 568.208,Z 265.914,A -85,B 0,C 180,E1 -1342.237,E2 -1342.237} C_VEL
LIN {X 0,Y 570.584,Z 274.579,A -85,B 0,C 180,E1 -1343.054,E2 -1343.054} C_VEL
LIN {X 0,Y 570.58,Z 314.764,A -85,B 0,C 180,E1 -1346.131,E2 -1346.131} C_VEL
LIN {X 0,Y 570.343,Z 356.327,A -85,B 0,C 180,E1 -1349.296,E2 -1349.296} C_VEL
LIN {X 0,Y 569.832,Z 396.228,A -85,B 0,C 180,E1 -1352.362,E2 -1352.362} C_VEL
LIN {X 0,Y 569.309,Z 440.162,A -85,B 0,C 180,E1 -1355.694,E2 -1355.694} C_VEL
LIN {X 0,Y 569.015,Z 472.31,A -85,B 0,C 180,E1 -1358.08,E2 -1358.08} C_VEL
LIN {X 0,Y 569.493,Z 479.62,A -85,B 0,C 180,E1 -1358.203,E2 -1358.203} C_VEL
LIN {X 0,Y 569.149,Z 615.458,A -85,B 0,C 180,E1 -1359.967,E2 -1359.967} C_VEL
LIN {X 0,Y 569.049,Z 632.104,A -85,B 0,C 180,E1 -1360.384,E2 -1360.384} C_VEL
LIN {X 0,Y 568.896,Z 647.047,A -85,B 0,C 180,E1 -1360.941,E2 -1360.941} C_VEL
LIN {X 0,Y 568.703,Z 662.249,A -85,B 0,C 180,E1 -1361.71,E2 -1361.71} C_VEL
LIN {X 0,Y 568.515,Z 676.52,A -85,B 0,C 180,E1 -1362.647,E2 -1362.647} C_VEL
LIN {X 0,Y 568.34,Z 689.626,A -85,B 0,C 180,E1 -1363.738,E2 -1363.738} C_VEL
LIN {X 0,Y 568.187,Z 701.677,A -85,B 0,C 180,E1 -1364.99,E2 -1364.99} C_VEL
LIN {X 0,Y 568.07,Z 712.106,A -85,B 0,C 180,E1 -1366.355,E2 -1366.355} C_VEL
LIN {X 0,Y 567.993,Z 721.041,A -85,B 0,C 180,E1 -1367.835,E2 -1367.835} C_VEL
LIN {X 0,Y 567.945,Z 727.94,A -85,B 0,C 180,E1 -1369.33,E2 -1369.33} C_VEL
LIN {X 0,Y 567.926,Z 733.391,A -85,B 0,C 180,E1 -1370.939,E2 -1370.939} C_VEL
LIN {X 0,Y 567.916,Z 736.958,A -85,B 0,C 180,E1 -1372.568,E2 -1372.568} C_VEL
LIN {X 0,Y 567.918,Z 738.756,A -85,B 0,C 180,E1 -1374.219,E2 -1374.219} C_VEL
LIN {X 0,Y 567.915,Z 738.818,A -85,B 0,C 180,E1 -1375.775,E2 -1375.775} C_VEL
LIN {X 0,Y 567.916,Z 737.039,A -85,B 0,C 180,E1 -1377.468,E2 -1377.468} C_VEL
LIN {X 0,Y 567.923,Z 733.621,A -85,B 0,C 180,E1 -1379.071,E2 -1379.071} C_VEL
LIN {X 0,Y 567.945,Z 728.188,A -85,B 0,C 180,E1 -1380.698,E2 -1380.698} C_VEL
LIN {X 0,Y 567.992,Z 721.158,A -85,B 0,C 180,E1 -1382.233,E2 -1382.233} C_VEL
LIN {X 0,Y 568.064,Z 712.542,A -85,B 0,C 180,E1 -1383.67,E2 -1383.67} C_VEL
LIN {X 0,Y 568.187,Z 701.789,A -85,B 0,C 180,E1 -1385.086,E2 -1385.086} C_VEL
LIN {X 0,Y 568.334,Z 690.011,A -85,B 0,C 180,E1 -1386.316,E2 -1386.316} C_VEL
LIN {X 0,Y 568.511,Z 677.153,A -85,B 0,C 180,E1 -1387.397,E2 -1387.397} C_VEL
LIN {X 0,Y 568.697,Z 662.595,A -85,B 0,C 180,E1 -1388.36,E2 -1388.36} C_VEL
LIN {X 0,Y 568.883,Z 647.742,A -85,B 0,C 180,E1 -1389.12,E2 -1389.12} C_VEL
LIN {X 0,Y 569.05,Z 631.274,A -85,B 0,C 180,E1 -1389.733,E2 -1389.733} C_VEL
LIN {X 0,Y 569.137,Z 614.862,A -85,B 0,C 180,E1 -1390.134,E2 -1390.134} C_VEL
LIN {X 0,Y 569.279,Z 474.786,A -85,B 0,C 180,E1 -1391.956,E2 -1391.956} C_VEL
LIN {X 0,Y 568.985,Z 472.015,A -85,B 0,C 180,E1 -1392.028,E2 -1392.028} C_VEL
LIN {X 0,Y 569.413,Z 430.843,A -85,B 0,C 180,E1 -1395.098,E2 -1395.098} C_VEL
LIN {X 0,Y 569.893,Z 388.518,A -85,B 0,C 180,E1 -1398.321,E2 -1398.321} C_VEL
LIN {X 0,Y 570.364,Z 352.171,A -85,B 0,C 180,E1 -1401.106,E2 -1401.106} C_VEL
LIN {X 0,Y 570.457,Z 309.748,A -85,B 0,C 180,E1 -1404.291,E2 -1404.291} C_VEL
LIN {X 0,Y 570.392,Z 279.968,A -85,B 0,C 180,E1 -1406.55,E2 -1406.55} C_VEL
LIN {X 0,Y 570.083,Z 272.371,A -85,B 0,C 180,E1 -1407.129,E2 -1407.129} C_VEL
LIN {X 0,Y 568.225,Z 266.024,A -85,B 0,C 180,E1 -1407.72,E2 -1407.72} C_VEL
LIN {X 0,Y 568.222,Z 265.707,A -85,B 0,C 180,E1 -1408.389,E2 -1408.389} C_VEL
LIN {X 0,Y 568.171,Z 265.708,A -85,B 0,C 180,E1 -1411.516,E2 -1411.516} C_VEL
LIN {X 0,Y 568.211,Z 265.705,A -85,B 0,C 180,E1 -1414.796,E2 -1414.796} C_VEL
LIN {X 0,Y 568.195,Z 265.71,A -85,B 0,C 180,E1 -1418.023,E2 -1418.023} C_VEL
LIN {X 0,Y 568.178,Z 265.704,A -85,B 0,C 180,E1 -1421.32,E2 -1421.32} C_VEL
LIN {X 0,Y 568.222,Z 265.706,A -85,B 0,C 180,E1 -1424.486,E2 -1424.486} C_VEL
LIN {X 0,Y 568.175,Z 265.707,A -85,B 0,C 180,E1 -1427.705,E2 -1427.705} C_VEL
LIN {X 0,Y 568.212,Z 265.702,A -85,B 0,C 180,E1 -1430.989,E2 -1430.989} C_VEL
LIN {X 0,Y 568.204,Z 265.709,A -85,B 0,C 180,E1 -1434.243,E2 -1434.243} C_VEL
LIN {X 0,Y 568.177,Z 265.705,A -85,B 0,C 180,E1 -1437.579,E2 -1437.579} C_VEL
LIN {X 0,Y 568.22,Z 265.704,A -85,B 0,C 180,E1 -1440.806,E2 -1440.806} C_VEL
LIN {X 0,Y 568.183,Z 265.707,A -85,B 0,C 180,E1 -1444.036,E2 -1444.036} C_VEL
LIN {X 0,Y 568.195,Z 265.702,A -85,B 0,C 180,E1 -1447.38,E2 -1447.38} C_VEL
LIN {X 0,Y 568.219,Z 265.708,A -85,B 0,C 180,E1 -1450.647,E2 -1450.647} C_VEL
LIN {X 0,Y 568.179,Z 265.705,A -85,B 0,C 180,E1 -1453.847,E2 -1453.847} C_VEL
LIN {X 0,Y 568.221,Z 265.702,A -85,B 0,C 180,E1 -1457.089,E2 -1457.089} C_VEL
LIN {X 0,Y 568.199,Z 265.708,A -85,B 0,C 180,E1 -1460.39,E2 -1460.39} C_VEL
LIN {X 0,Y 568.184,Z 265.704,A -85,B 0,C 180,E1 -1463.764,E2 -1463.764} C_VEL
LIN {X 0,Y 568.219,Z 265.704,A -85,B 0,C 180,E1 -1466.999,E2 -1466.999} C_VEL
LIN {X 0,Y 568.186,Z 265.706,A -85,B 0,C 180,E1 -1470.231,E2 -1470.231} C_VEL
LIN {X 0,Y 568.207,Z 265.701,A -85,B 0,C 180,E1 -1473.541,E2 -1473.541} C_VEL
LIN {X 0,Y 568.22,Z 265.708,A -85,B 0,C 180,E1 -1476.872,E2 -1476.872} C_VEL
LIN {X 0,Y 568.184,Z 265.705,A -85,B 0,C 180,E1 -1480.095,E2 -1480.095} C_VEL
LIN {X 0,Y 568.22,Z 265.703,A -85,B 0,C 180,E1 -1483.39,E2 -1483.39} C_VEL
LIN {X 0,Y 568.212,Z 265.709,A -85,B 0,C 180,E1 -1486.76,E2 -1486.76} C_VEL
LIN {X 0,Y 568.188,Z 265.705,A -85,B 0,C 180,E1 -1490.038,E2 -1490.038} C_VEL
LIN {X 0,Y 568.214,Z 265.69,A -85,B 0,C 180,E1 -1493.255,E2 -1493.255} C_VEL
LIN {X 0,Y 568.191,Z 265.706,A -85,B 0,C 180,E1 -1496.523,E2 -1496.523} C_VEL
LIN {X 0,Y 568.308,Z 266.324,A -85,B 0,C 180,E1 -1496.762,E2 -1496.762} C_VEL
LIN {X 0,Y 572.185,Z 277.197,A -85,B 0,C 180,E1 -1497.796,E2 -1497.796} C_VEL
LIN {X 0,Y 571.647,Z 315.823,A -85,B 0,C 180,E1 -1500.395,E2 -1500.395} C_VEL
LIN {X 0,Y 572.659,Z 323.284,A -85,B 0,C 180,E1 -1500.561,E2 -1500.561} C_VEL
LIN {X 0,Y 571.734,Z 552.304,A -85,B 0,C 180,E1 -1503.698,E2 -1503.698} C_VEL
